  MoveL 10629 to (234.05, 162.02, 144.49) mm, rotated rx 180 ry 0 rz 180 deg; joints [-145.976, -74.933, -32.212, 66.411, 37.63, -61.13]
  Call Extruder(657.74297)
  MoveL 10630 to (233.75, 162.2, 144.49) mm, rotated rx -180 ry 0 rz 180 deg; joints [-145.947, -74.903, -32.271, 66.399, 37.667, -61.104]
  MoveL 10631 to (233.75, 162.2, 144.49) mm, rotated rx -180 ry 0 rz 180 deg; joints [-145.947, -74.903, -32.271, 66.399, 37.667, -61.104]
  Call Extruder(657.94993)
  MoveL 10632 to (233.45, 162.37, 144.49) mm, rotated rx 180 ry 0 rz 180 deg; joints [-145.919, -74.874, -32.33, 66.387, 37.703, -61.078]
  MoveL 10633 to (233.45, 162.37, 144.49) mm, rotated rx 180 ry 0 rz 180 deg; joints [-145.919, -74.874, -32.33, 66.387, 37.703, -61.078]
  Call Extruder(658.15610)
  MoveL 10634 to (233.14, 162.55, 144.49) mm, rotated rx 180 ry 0 rz 180 deg; joints [-145.89, -74.844, -32.388, 66.376, 37.74, -61.053]
  MoveL 10635 to (233.14, 162.55, 144.49) mm, rotated rx 180 ry 0 rz 180 deg; joints [-145.89, -74.844, -32.388, 66.376, 37.74, -61.053]
  Call Extruder(658.33777)
  MoveL 10636 to (232.87, 162.69, 144.49) mm, rotated rx 180 ry 0 rz 180 deg; joints [-145.866, -74.815, -32.446, 66.361, 37.772, -61.026]
  MoveL 10637 to (232.87, 162.69, 144.49) mm, rotated rx 180 ry 0 rz 180 deg; joints [-145.866, -74.815, -32.446, 66.361, 37.772, -61.026]
  Call Extruder(658.49574)
  MoveL 10638 to (232.62, 162.8, 144.49) mm, rotated rx -180 ry 0 rz -180 deg; joints [-145.845, -74.787, -32.501, 66.345, 37.801, -60.997]
  MoveL 10639 to (232.62, 162.8, 144.49) mm, rotated rx -180 ry 0 rz -180 deg; joints [-145.845, -74.787, -32.501, 66.345, 37.801, -60.997]
  Call Extruder(658.65309)
  MoveL 10640 to (232.37, 162.91, 144.49) mm, rotated rx -180 ry 0 rz 180 deg; joints [-145.825, -74.759, -32.557, 66.329, 37.83, -60.969]
  MoveL 10641 to (232.37, 162.91, 144.49) mm, rotated rx -180 ry 0 rz 180 deg; joints [-145.825, -74.759, -32.557, 66.329, 37.83, -60.969]
  Call Extruder(658.83583)
  MoveL 10642 to (232.07, 163.02, 144.49) mm, rotated rx 180 ry 0 rz 180 deg; joints [-145.801, -74.725, -32.623, 66.309, 37.864, -60.935]
  MoveL 10643 to (232.07, 163.02, 144.49) mm, rotated rx 180 ry 0 rz 180 deg; joints [-145.801, -74.725, -32.623, 66.309, 37.864, -60.935]
  Call Extruder(659.01781)
  MoveL 10644 to (231.78, 163.15, 144.49) mm, rotated rx -180 ry 0 rz 180 deg; joints [-145.777, -74.692, -32.689, 66.29, 37.898, -60.901]
  MoveL 10645 to (231.78, 163.15, 144.49) mm, rotated rx -180 ry 0 rz 180 deg; joints [-145.777, -74.692, -32.689, 66.29, 37.898, -60.901]
  Call Extruder(659.16515)
  MoveL 10646 to (231.54, 163.24, 144.49) mm, rotated rx -180 ry 0 rz -180 deg; joints [-145.759, -74.664, -32.745, 66.272, 37.926, -60.872]
  MoveL 10647 to (231.54, 163.24, 144.49) mm, rotated rx -180 ry 0 rz -180 deg; joints [-145.759, -74.664, -32.745, 66.272, 37.926, -60.872]
  Call Extruder(659.27837)
  MoveL 10648 to (231.35, 163.3, 144.49) mm, rotated rx -180 ry 0 rz 180 deg; joints [-145.744, -74.641, -32.791, 66.257, 37.947, -60.847]
  MoveL 10649 to (231.35, 163.3, 144.49) mm, rotated rx -180 ry 0 rz 180 deg; joints [-145.744, -74.641, -32.791, 66.257, 37.947, -60.847]
  Call Extruder(659.39115)
  MoveL 10650 to (231.17, 163.36, 144.49) mm, rotated rx 180 ry 0 rz 180 deg; joints [-145.73, -74.618, -32.836, 66.241, 37.969, -60.822]
  MoveL 10651 to (231.17, 163.36, 144.49) mm, rotated rx 180 ry 0 rz 180 deg; joints [-145.73, -74.618, -32.836, 66.241, 37.969, -60.822]
  Call Extruder(659.50349)
  MoveL 10652 to (230.98, 163.42, 144.49) mm, rotated rx 180 ry 0 rz 180 deg; joints [-145.716, -74.594, -32.882, 66.226, 37.99, -60.797]
  MoveL 10653 to (230.98, 163.42, 144.49) mm, rotated rx 180 ry 0 rz 180 deg; joints [-145.716, -74.594, -32.882, 66.226, 37.99, -60.797]
  Call Extruder(659.61538)
  MoveL 10654 to (230.79, 163.48, 144.49) mm, rotated rx 180 ry 0 rz 180 deg; joints [-145.702, -74.571, -32.928, 66.21, 38.012, -60.772]
  MoveL 10655 to (230.79, 163.48, 144.49) mm, rotated rx 180 ry 0 rz 180 deg; joints [-145.702, -74.571, -32.928, 66.21, 38.012, -60.772]
  Call Extruder(659.73678)
  MoveL 10656 to (230.58, 163.55, 144.49) mm, rotated rx 180 ry 0 rz 180 deg; joints [-145.687, -74.546, -32.978, 66.193, 38.035, -60.745]
  MoveL 10657 to (230.58, 163.55, 144.49) mm, rotated rx 180 ry 0 rz 180 deg; joints [-145.687, -74.546, -32.978, 66.193, 38.035, -60.745]
  Call Extruder(659.86760)
  MoveL 10658 to (230.36, 163.61, 144.49) mm, rotated rx 180 ry 0 rz 180 deg; joints [-145.67, -74.518, -33.034, 66.174, 38.06, -60.714]
  MoveL 10659 to (230.36, 163.61, 144.49) mm, rotated rx 180 ry 0 rz 180 deg; joints [-145.67, -74.518, -33.034, 66.174, 38.06, -60.714]
  Call Extruder(659.99784)
  MoveL 10660 to (230.14, 163.68, 144.49) mm, rotated rx 180 ry 0 rz 180 deg; joints [-145.654, -74.49, -33.089, 66.155, 38.086, -60.684]
  MoveL 10661 to (230.14, 163.68, 144.49) mm, rotated rx 180 ry 0 rz 180 deg; joints [-145.654, -74.49, -33.089, 66.155, 38.086, -60.684]
  Call Extruder(660.12753)
  MoveL 10662 to (229.91, 163.75, 144.49) mm, rotated rx 180 ry 0 rz 180 deg; joints [-145.638, -74.462, -33.144, 66.137, 38.111, -60.654]
  MoveL 10663 to (229.91, 163.75, 144.49) mm, rotated rx 180 ry 0 rz 180 deg; joints [-145.638, -74.462, -33.144, 66.137, 38.111, -60.654]
  Call Extruder(660.25665)
  MoveL 10664 to (229.69, 163.82, 144.49) mm, rotated rx -180 ry 0 rz 180 deg; joints [-145.621, -74.434, -33.199, 66.118, 38.136, -60.624]
  MoveL 10665 to (229.69, 163.82, 144.49) mm, rotated rx -180 ry 0 rz 180 deg; joints [-145.621, -74.434, -33.199, 66.118, 38.136, -60.624]
  Call Extruder(660.37172)
  MoveL 10666 to (229.48, 163.86, 144.49) mm, rotated rx 180 ry 0 rz -180 deg; joints [-145.607, -74.407, -33.253, 66.098, 38.159, -60.593]
  MoveL 10667 to (229.48, 163.86, 144.49) mm, rotated rx 180 ry 0 rz -180 deg; joints [-145.607, -74.407, -33.253, 66.098, 38.159, -60.593]
  Call Extruder(660.48634)
  MoveL 10668 to (229.28, 163.91, 144.49) mm, rotated rx 180 ry 0 rz -180 deg; joints [-145.594, -74.38, -33.306, 66.078, 38.182, -60.562]
  MoveL 10669 to (229.28, 163.91, 144.49) mm, rotated rx 180 ry 0 rz -180 deg; joints [-145.594, -74.38, -33.306, 66.078, 38.182, -60.562]
  Call Extruder(660.60051)
  MoveL 10670 to (229.08, 163.95, 144.49) mm, rotated rx 180 ry 0 rz 180 deg; joints [-145.58, -74.353, -33.36, 66.058, 38.204, -60.532]
  MoveL 10671 to (229.08, 163.95, 144.49) mm, rotated rx 180 ry 0 rz 180 deg; joints [-145.58, -74.353, -33.36, 66.058, 38.204, -60.532]
  Call Extruder(660.71423)
  MoveL 10672 to (228.87, 164, 144.49) mm, rotated rx -180 ry 0 rz -180 deg; joints [-145.566, -74.326, -33.414, 66.038, 38.227, -60.501]
  MoveL 10673 to (228.87, 164, 144.49) mm, rotated rx -180 ry 0 rz -180 deg; joints [-145.566, -74.326, -33.414, 66.038, 38.227, -60.501]
  Call Extruder(660.83965)
  MoveL 10674 to (228.65, 164.04, 144.49) mm, rotated rx 180 ry 0 rz -180 deg; joints [-145.551, -74.296, -33.473, 66.016, 38.252, -60.467]
  MoveL 10675 to (228.65, 164.04, 144.49) mm, rotated rx 180 ry 0 rz -180 deg; joints [-145.551, -74.296, -33.473, 66.016, 38.252, -60.467]
  Call Extruder(660.97663)
  MoveL 10676 to (228.4, 164.09, 144.49) mm, rotated rx 180 ry 0 rz 180 deg; joints [-145.535, -74.263, -33.539, 65.991, 38.28, -60.429]
  MoveL 10677 to (228.4, 164.09, 144.49) mm, rotated rx 180 ry 0 rz 180 deg; joints [-145.535, -74.263, -33.539, 65.991, 38.28, -60.429]
  Call Extruder(661.11299)
  MoveL 10678 to (228.15, 164.14, 144.49) mm, rotated rx 180 ry 0 rz 180 deg; joints [-145.518, -74.229, -33.606, 65.966, 38.308, -60.391]
  MoveL 10679 to (228.15, 164.14, 144.49) mm, rotated rx 180 ry 0 rz 180 deg; joints [-145.518, -74.229, -33.606, 65.966, 38.308, -60.391]
  Call Extruder(661.24875)
  MoveL 10680 to (227.9, 164.19, 144.49) mm, rotated rx 180 ry 0 rz 180 deg; joints [-145.502, -74.196, -33.672, 65.942, 38.335, -60.353]
  MoveL 10681 to (227.9, 164.19, 144.49) mm, rotated rx 180 ry 0 rz 180 deg; joints [-145.502, -74.196, -33.672, 65.942, 38.335, -60.353]
  Call Extruder(661.38390)
  MoveL 10682 to (227.65, 164.24, 144.49) mm, rotated rx 180 ry 0 rz -180 deg; joints [-145.485, -74.163, -33.738, 65.917, 38.363, -60.315]
  MoveL 10683 to (227.65, 164.24, 144.49) mm, rotated rx 180 ry 0 rz -180 deg; joints [-145.485, -74.163, -33.738, 65.917, 38.363, -60.315]
  Call Extruder(661.51844)
  MoveL 10684 to (227.4, 164.29, 144.49) mm, rotated rx -180 ry 0 rz 180 deg; joints [-145.469, -74.129, -33.803, 65.893, 38.39, -60.278]
  MoveL 10685 to (227.4, 164.29, 144.49) mm, rotated rx -180 ry 0 rz 180 deg; joints [-145.469, -74.129, -33.803, 65.893, 38.39, -60.278]
  Call Extruder(661.65236)
  MoveL 10686 to (227.15, 164.34, 144.49) mm, rotated rx -180 ry 0 rz -180 deg; joints [-145.453, -74.096, -33.869, 65.868, 38.418, -60.24]
  MoveL 10687 to (227.15, 164.34, 144.49) mm, rotated rx -180 ry 0 rz -180 deg; joints [-145.453, -74.096, -33.869, 65.868, 38.418, -60.24]
  Call Extruder(661.80023)
  MoveL 10688 to (226.87, 164.39, 144.49) mm, rotated rx 180 ry 0 rz -180 deg; joints [-145.435, -74.059, -33.943, 65.84, 38.448, -60.197]
  MoveL 10689 to (226.87, 164.39, 144.49) mm, rotated rx 180 ry 0 rz -180 deg; joints [-145.435, -74.059, -33.943, 65.84, 38.448, -60.197]
  Call Extruder(661.96197)
  MoveL 10690 to (226.57, 164.44, 144.49) mm, rotated rx 180 ry 0 rz 180 deg; joints [-145.415, -74.017, -34.026, 65.809, 38.482, -60.149]
  MoveL 10691 to (226.57, 164.44, 144.49) mm, rotated rx 180 ry 0 rz 180 deg; joints [-145.415, -74.017, -34.026, 65.809, 38.482, -60.149]
  Call Extruder(662.12298)
  MoveL 10692 to (226.26, 164.49, 144.49) mm, rotated rx -180 ry 0 rz 180 deg; joints [-145.396, -73.975, -34.109, 65.777, 38.516, -60.101]
  MoveL 10693 to (226.26, 164.49, 144.49) mm, rotated rx -180 ry 0 rz 180 deg; joints [-145.396, -73.975, -34.109, 65.777, 38.516, -60.101]
  Call Extruder(662.28327)
  MoveL 10694 to (225.95, 164.53, 144.49) mm, rotated rx -180 ry 0 rz 180 deg; joints [-145.377, -73.934, -34.191, 65.746, 38.549, -60.054]
  MoveL 10695 to (225.95, 164.53, 144.49) mm, rotated rx -180 ry 0 rz 180 deg; joints [-145.377, -73.934, -34.191, 65.746, 38.549, -60.054]
  Call Extruder(662.44282)
  MoveL 10696 to (225.65, 164.58, 144.49) mm, rotated rx -180 ry 0 rz 180 deg; joints [-145.357, -73.892, -34.273, 65.715, 38.583, -60.006]
  MoveL 10697 to (225.65, 164.58, 144.49) mm, rotated rx -180 ry 0 rz 180 deg; joints [-145.357, -73.892, -34.273, 65.715, 38.583, -60.006]
  Call Extruder(662.60165)
  MoveL 10698 to (225.34, 164.63, 144.49) mm, rotated rx -180 ry 0 rz 180 deg; joints [-145.338, -73.851, -34.355, 65.684, 38.616, -59.959]
  MoveL 10699 to (225.34, 164.63, 144.49) mm, rotated rx -180 ry 0 rz 180 deg; joints [-145.338, -73.851, -34.355, 65.684, 38.616, -59.959]
  Call Extruder(662.78032)
  MoveL 10700 to (225, 164.68, 144.49) mm, rotated rx 180 ry 0 rz 180 deg; joints [-145.317, -73.803, -34.45, 65.647, 38.654, -59.904]
  MoveL 10701 to (225, 164.68, 144.49) mm, rotated rx 180 ry 0 rz 180 deg; joints [-145.317, -73.803, -34.45, 65.647, 38.654, -59.904]
  Call Extruder(662.97876)
  MoveL 10702 to (224.61, 164.72, 144.49) mm, rotated rx -180 ry 0 rz 180 deg; joints [-145.293, -73.749, -34.557, 65.606, 38.696, -59.841]
  MoveL 10703 to (224.61, 164.72, 144.49) mm, rotated rx -180 ry 0 rz 180 deg; joints [-145.293, -73.749, -34.557, 65.606, 38.696, -59.841]
  Call Extruder(663.17634)
  MoveL 10704 to (224.22, 164.77, 144.49) mm, rotated rx 180 ry 0 rz 180 deg; joints [-145.27, -73.696, -34.664, 65.565, 38.738, -59.779]
  MoveL 10705 to (224.22, 164.77, 144.49) mm, rotated rx 180 ry 0 rz 180 deg; joints [-145.27, -73.696, -34.664, 65.565, 38.738, -59.779]
  Call Extruder(663.37305)
  MoveL 10706 to (223.83, 164.82, 144.49) mm, rotated rx 180 ry 0 rz 180 deg; joints [-145.246, -73.642, -34.77, 65.524, 38.78, -59.717]
  MoveL 10707 to (223.83, 164.82, 144.49) mm, rotated rx 180 ry 0 rz 180 deg; joints [-145.246, -73.642, -34.77, 65.524, 38.78, -59.717]
  Call Extruder(663.56888)
  MoveL 10708 to (223.45, 164.86, 144.49) mm, rotated rx 180 ry 0 rz 180 deg; joints [-145.223, -73.588, -34.876, 65.483, 38.823, -59.655]
  MoveL 10709 to (223.45, 164.86, 144.49) mm, rotated rx 180 ry 0 rz 180 deg; joints [-145.223, -73.588, -34.876, 65.483, 38.823, -59.655]
  Call Extruder(663.86424)
  MoveL 10710 to (222.86, 164.91, 144.49) mm, rotated rx 180 ry 0 rz -180 deg; joints [-145.189, -73.505, -35.042, 65.418, 38.886, -59.557]
  MoveL 10711 to (222.86, 164.91, 144.49) mm, rotated rx 180 ry 0 rz -180 deg; joints [-145.189, -73.505, -35.042, 65.418, 38.886, -59.557]
  Call Extruder(664.15827)
  MoveL 10712 to (222.27, 164.95, 144.49) mm, rotated rx 180 ry 0 rz 180 deg; joints [-145.155, -73.422, -35.207, 65.353, 38.949, -59.46]
  MoveL 10713 to (222.27, 164.95, 144.49) mm, rotated rx 180 ry 0 rz 180 deg; joints [-145.155, -73.422, -35.207, 65.353, 38.949, -59.46]
  Call Extruder(664.45096)
  MoveL 10714 to (221.68, 165, 144.49) mm, rotated rx 180 ry 0 rz 180 deg; joints [-145.121, -73.339, -35.371, 65.289, 39.013, -59.364]
  MoveL 10715 to (221.68, 165, 144.49) mm, rotated rx 180 ry 0 rz 180 deg; joints [-145.121, -73.339, -35.371, 65.289, 39.013, -59.364]
  Call Extruder(665.02441)
  MoveL 10716 to (220.52, 165.05, 144.49) mm, rotated rx 180 ry 0 rz 180 deg; joints [-145.056, -73.172, -35.703, 65.157, 39.137, -59.167]
  MoveL 10717 to (220.52, 165.05, 144.49) mm, rotated rx 180 ry 0 rz 180 deg; joints [-145.056, -73.172, -35.703, 65.157, 39.137, -59.167]
  Call Extruder(665.73842)
  MoveL 10718 to (219.06, 165.09, 144.49) mm, rotated rx 180 ry 0 rz 180 deg; joints [-144.977, -72.963, -36.118, 64.992, 39.292, -58.921]
  Call Extruder(782.58519)
  MoveL 10719 to (-19.06, 165.09, 144.49) mm, rotated rx -180 ry 0 rz 180 deg; joints [-127.435, -51.662, -80.11, 62.98, 63.042, -41.636]
  Call Extruder(783.01380)
  MoveL 10720 to (-19.94, 165.07, 144.49) mm, rotated rx 180 ry 0 rz 180 deg; joints [-127.348, -51.612, -80.219, 63.026, 63.126, -41.61]
  MoveL 10721 to (-19.94, 165.07, 144.49) mm, rotated rx 180 ry 0 rz 180 deg; joints [-127.348, -51.612, -80.219, 63.026, 63.126, -41.61]
  Call Extruder(783.58725)
  MoveL 10722 to (-21.1, 165.02, 144.49) mm, rotated rx -180 ry 0 rz 180 deg; joints [-127.235, -51.545, -80.367, 63.085, 63.238, -41.573]
  MoveL 10723 to (-21.1, 165.02, 144.49) mm, rotated rx -180 ry 0 rz 180 deg; joints [-127.235, -51.545, -80.367, 63.085, 63.238, -41.573]
  Call Extruder(784.02155)
  MoveL 10724 to (-21.97, 164.98, 144.49) mm, rotated rx 180 ry 0 rz 180 deg; joints [-127.15, -51.493, -80.48, 63.129, 63.322, -41.543]
  MoveL 10725 to (-21.97, 164.98, 144.49) mm, rotated rx 180 ry 0 rz 180 deg; joints [-127.15, -51.493, -80.48, 63.129, 63.322, -41.543]
  Call Extruder(784.31557)
  MoveL 10726 to (-22.56, 164.93, 144.49) mm, rotated rx 180 ry 0 rz 180 deg; joints [-127.093, -51.457, -80.558, 63.157, 63.378, -41.522]
  MoveL 10727 to (-22.56, 164.93, 144.49) mm, rotated rx 180 ry 0 rz 180 deg; joints [-127.093, -51.457, -80.558, 63.157, 63.378, -41.522]
  Call Extruder(784.61093)
  MoveL 10728 to (-23.15, 164.89, 144.49) mm, rotated rx 180 ry 0 rz 180 deg; joints [-127.037, -51.421, -80.636, 63.185, 63.435, -41.501]
  MoveL 10729 to (-23.15, 164.89, 144.49) mm, rotated rx 180 ry 0 rz 180 deg; joints [-127.037, -51.421, -80.636, 63.185, 63.435, -41.501]
  Call Extruder(784.85715)
  MoveL 10730 to (-23.64, 164.84, 144.49) mm, rotated rx 180 ry 0 rz 180 deg; joints [-126.991, -51.391, -80.702, 63.207, 63.481, -41.482]
  MoveL 10731 to (-23.64, 164.84, 144.49) mm, rotated rx 180 ry 0 rz 180 deg; joints [-126.991, -51.391, -80.702, 63.207, 63.481, -41.482]
  Call Extruder(785.05385)
  MoveL 10732 to (-24.03, 164.79, 144.49) mm, rotated rx -180 ry 0 rz 180 deg; joints [-126.955, -51.367, -80.756, 63.224, 63.518, -41.467]
  MoveL 10733 to (-24.03, 164.79, 144.49) mm, rotated rx -180 ry 0 rz 180 deg; joints [-126.955, -51.367, -80.756, 63.224, 63.518, -41.467]
  Call Extruder(785.25143)
  MoveL 10734 to (-24.42, 164.75, 144.49) mm, rotated rx -180 ry 0 rz 180 deg; joints [-126.919, -51.342, -80.81, 63.242, 63.555, -41.451]
  MoveL 10735 to (-24.42, 164.75, 144.49) mm, rotated rx -180 ry 0 rz 180 deg; joints [-126.919, -51.342, -80.81, 63.242, 63.555, -41.451]
  Call Extruder(785.44987)
  MoveL 10736 to (-24.8, 164.7, 144.49) mm, rotated rx -180 ry 0 rz 180 deg; joints [-126.883, -51.318, -80.863, 63.259, 63.592, -41.435]
  MoveL 10737 to (-24.8, 164.7, 144.49) mm, rotated rx -180 ry 0 rz 180 deg; joints [-126.883, -51.318, -80.863, 63.259, 63.592, -41.435]
  Call Extruder(785.64918)
  MoveL 10738 to (-25.19, 164.66, 144.49) mm, rotated rx 180 ry 0 rz 180 deg; joints [-126.847, -51.293, -80.917, 63.276, 63.629, -41.42]
  MoveL 10739 to (-25.19, 164.66, 144.49) mm, rotated rx 180 ry 0 rz 180 deg; joints [-126.847, -51.293, -80.917, 63.276, 63.629, -41.42]
  Call Extruder(785.80801)
  MoveL 10740 to (-25.5, 164.61, 144.49) mm, rotated rx -180 ry 0 rz 180 deg; joints [-126.82, -51.273, -80.961, 63.288, 63.658, -41.406]
  MoveL 10741 to (-25.5, 164.61, 144.49) mm, rotated rx -180 ry 0 rz 180 deg; joints [-126.82, -51.273, -80.961, 63.288, 63.658, -41.406]
  Call Extruder(785.96757)
  MoveL 10742 to (-25.8, 164.56, 144.49) mm, rotated rx 180 ry 0 rz 180 deg; joints [-126.792, -51.253, -81.005, 63.301, 63.687, -41.393]
  MoveL 10743 to (-25.8, 164.56, 144.49) mm, rotated rx 180 ry 0 rz 180 deg; joints [-126.792, -51.253, -81.005, 63.301, 63.687, -41.393]
  Call Extruder(786.12786)
  MoveL 10744 to (-26.11, 164.51, 144.49) mm, rotated rx 180 ry 0 rz -180 deg; joints [-126.765, -51.233, -81.049, 63.313, 63.716, -41.379]
  MoveL 10745 to (-26.11, 164.51, 144.49) mm, rotated rx 180 ry 0 rz -180 deg; joints [-126.765, -51.233, -81.049, 63.313, 63.716, -41.379]
  Call Extruder(786.28887)
  MoveL 10746 to (-26.41, 164.46, 144.49) mm, rotated rx -180 ry 0 rz 180 deg; joints [-126.737, -51.213, -81.093, 63.326, 63.745, -41.365]
  MoveL 10747 to (-26.41, 164.46, 144.49) mm, rotated rx -180 ry 0 rz 180 deg; joints [-126.737, -51.213, -81.093, 63.326, 63.745, -41.365]
  Call Extruder(786.45061)
  MoveL 10748 to (-26.72, 164.41, 144.49) mm, rotated rx 180 ry 0 rz 180 deg; joints [-126.71, -51.193, -81.137, 63.338, 63.774, -41.352]
  MoveL 10749 to (-26.72, 164.41, 144.49) mm, rotated rx 180 ry 0 rz 180 deg; joints [-126.71, -51.193, -81.137, 63.338, 63.774, -41.352]
  Call Extruder(786.61308)
  MoveL 10750 to (-27.03, 164.36, 144.49) mm, rotated rx 180 ry 0 rz 180 deg; joints [-126.682, -51.172, -81.181, 63.351, 63.803, -41.338]
  MoveL 10751 to (-27.03, 164.36, 144.49) mm, rotated rx 180 ry 0 rz 180 deg; joints [-126.682, -51.172, -81.181, 63.351, 63.803, -41.338]
  Call Extruder(786.74701)
  MoveL 10752 to (-27.27, 164.32, 144.49) mm, rotated rx -180 ry 0 rz 180 deg; joints [-126.66, -51.155, -81.218, 63.36, 63.826, -41.326]
  MoveL 10753 to (-27.27, 164.32, 144.49) mm, rotated rx -180 ry 0 rz 180 deg; joints [-126.66, -51.155, -81.218, 63.36, 63.826, -41.326]
  Call Extruder(786.88155)
  MoveL 10754 to (-27.52, 164.27, 144.49) mm, rotated rx -180 ry 0 rz -180 deg; joints [-126.638, -51.138, -81.256, 63.37, 63.85, -41.314]
  MoveL 10755 to (-27.52, 164.27, 144.49) mm, rotated rx -180 ry 0 rz -180 deg; joints [-126.638, -51.138, -81.256, 63.37, 63.85, -41.314]
  Call Extruder(787.01669)
  MoveL 10756 to (-27.77, 164.22, 144.49) mm, rotated rx -180 ry 0 rz 180 deg; joints [-126.617, -51.121, -81.293, 63.379, 63.873, -41.301]
  MoveL 10757 to (-27.77, 164.22, 144.49) mm, rotated rx -180 ry 0 rz 180 deg; joints [-126.617, -51.121, -81.293, 63.379, 63.873, -41.301]
  Call Extruder(787.15245)
  MoveL 10758 to (-28.02, 164.17, 144.49) mm, rotated rx 180 ry 0 rz 180 deg; joints [-126.595, -51.104, -81.33, 63.388, 63.897, -41.289]
  MoveL 10759 to (-28.02, 164.17, 144.49) mm, rotated rx 180 ry 0 rz 180 deg; joints [-126.595, -51.104, -81.33, 63.388, 63.897, -41.289]
  Call Extruder(787.28882)
  MoveL 10760 to (-28.27, 164.12, 144.49) mm, rotated rx -180 ry 0 rz -180 deg; joints [-126.573, -51.087, -81.368, 63.398, 63.92, -41.277]
  MoveL 10761 to (-28.27, 164.12, 144.49) mm, rotated rx -180 ry 0 rz -180 deg; joints [-126.573, -51.087, -81.368, 63.398, 63.92, -41.277]
  Call Extruder(787.42580)
  MoveL 10762 to (-28.52, 164.07, 144.49) mm, rotated rx -180 ry 0 rz -180 deg; joints [-126.551, -51.07, -81.405, 63.407, 63.944, -41.265]
  MoveL 10763 to (-28.52, 164.07, 144.49) mm, rotated rx -180 ry 0 rz -180 deg; joints [-126.551, -51.07, -81.405, 63.407, 63.944, -41.265]
  Call Extruder(787.56338)
  MoveL 10764 to (-28.77, 164.02, 144.49) mm, rotated rx 180 ry 0 rz -180 deg; joints [-126.529, -51.053, -81.442, 63.417, 63.967, -41.253]
  MoveL 10765 to (-28.77, 164.02, 144.49) mm, rotated rx 180 ry 0 rz -180 deg; joints [-126.529, -51.053, -81.442, 63.417, 63.967, -41.253]
  Call Extruder(787.67710)
  MoveL 10766 to (-28.97, 163.97, 144.49) mm, rotated rx -180 ry 0 rz 180 deg; joints [-126.511, -51.039, -81.473, 63.424, 63.987, -41.243]
  MoveL 10767 to (-28.97, 163.97, 144.49) mm, rotated rx -180 ry 0 rz 180 deg; joints [-126.511, -51.039, -81.473, 63.424, 63.987, -41.243]
  Call Extruder(787.79127)
  MoveL 10768 to (-29.18, 163.93, 144.49) mm, rotated rx -180 ry 0 rz -180 deg; joints [-126.494, -51.025, -81.504, 63.431, 64.006, -41.232]
  MoveL 10769 to (-29.18, 163.93, 144.49) mm, rotated rx -180 ry 0 rz -180 deg; joints [-126.494, -51.025, -81.504, 63.431, 64.006, -41.232]
  Call Extruder(787.90589)
  MoveL 10770 to (-29.38, 163.88, 144.49) mm, rotated rx 180 ry 0 rz 180 deg; joints [-126.476, -51.011, -81.535, 63.439, 64.025, -41.222]
  MoveL 10771 to (-29.38, 163.88, 144.49) mm, rotated rx 180 ry 0 rz 180 deg; joints [-126.476, -51.011, -81.535, 63.439, 64.025, -41.222]
  Call Extruder(788.02096)
  MoveL 10772 to (-29.59, 163.84, 144.49) mm, rotated rx 180 ry 0 rz 180 deg; joints [-126.459, -50.997, -81.566, 63.446, 64.044, -41.211]
  MoveL 10773 to (-29.59, 163.84, 144.49) mm, rotated rx 180 ry 0 rz 180 deg; joints [-126.459, -50.997, -81.566, 63.446, 64.044, -41.211]
  Call Extruder(788.14320)
  MoveL 10774 to (-29.8, 163.78, 144.49) mm, rotated rx -180 ry 0 rz 180 deg; joints [-126.441, -50.981, -81.6, 63.453, 64.064, -41.2]
  MoveL 10775 to (-29.8, 163.78, 144.49) mm, rotated rx -180 ry 0 rz 180 deg; joints [-126.441, -50.981, -81.6, 63.453, 64.064, -41.2]
  Call Extruder(788.27288)
  MoveL 10776 to (-30.02, 163.72, 144.49) mm, rotated rx 180 ry 0 rz -180 deg; joints [-126.423, -50.964, -81.638, 63.459, 64.085, -41.186]
  MoveL 10777 to (-30.02, 163.72, 144.49) mm, rotated rx 180 ry 0 rz -180 deg; joints [-126.423, -50.964, -81.638, 63.459, 64.085, -41.186]
  Call Extruder(788.40312)
  MoveL 10778 to (-30.25, 163.65, 144.49) mm, rotated rx -180 ry 0 rz 180 deg; joints [-126.405, -50.947, -81.675, 63.466, 64.106, -41.173]
  MoveL 10779 to (-30.25, 163.65, 144.49) mm, rotated rx -180 ry 0 rz 180 deg; joints [-126.405, -50.947, -81.675, 63.466, 64.106, -41.173]
  Call Extruder(788.53393)
  MoveL 10780 to (-30.47, 163.58, 144.49) mm, rotated rx 180 ry 0 rz -180 deg; joints [-126.387, -50.931, -81.711, 63.472, 64.127, -41.159]
  MoveL 10781 to (-30.47, 163.58, 144.49) mm, rotated rx 180 ry 0 rz -180 deg; joints [-126.387, -50.931, -81.711, 63.472, 64.127, -41.159]
  Call Extruder(788.66530)
  MoveL 10782 to (-30.69, 163.51, 144.49) mm, rotated rx -180 ry 0 rz -180 deg; joints [-126.369, -50.914, -81.748, 63.478, 64.148, -41.146]
  MoveL 10783 to (-30.69, 163.51, 144.49) mm, rotated rx -180 ry 0 rz -180 deg; joints [-126.369, -50.914, -81.748, 63.478, 64.148, -41.146]
  Call Extruder(788.77719)
  MoveL 10784 to (-30.88, 163.45, 144.49) mm, rotated rx 180 ry 0 rz -180 deg; joints [-126.354, -50.899, -81.78, 63.483, 64.165, -41.134]
  MoveL 10785 to (-30.88, 163.45, 144.49) mm, rotated rx 180 ry 0 rz -180 deg; joints [-126.354, -50.899, -81.78, 63.483, 64.165, -41.134]
  Call Extruder(788.88953)
  MoveL 10786 to (-31.07, 163.39, 144.49) mm, rotated rx 180 ry 0 rz 180 deg; joints [-126.339, -50.885, -81.812, 63.488, 64.183, -41.122]
  MoveL 10787 to (-31.07, 163.39, 144.49) mm, rotated rx 180 ry 0 rz 180 deg; joints [-126.339, -50.885, -81.812, 63.488, 64.183, -41.122]
  Call Extruder(789.00231)
  MoveL 10788 to (-31.26, 163.33, 144.49) mm, rotated rx 180 ry 0 rz 180 deg; joints [-126.324, -50.87, -81.844, 63.493, 64.2, -41.11]
  MoveL 10789 to (-31.26, 163.33, 144.49) mm, rotated rx 180 ry 0 rz 180 deg; joints [-126.324, -50.87, -81.844, 63.493, 64.2, -41.11]
  Call Extruder(789.11553)
  MoveL 10790 to (-31.45, 163.27, 144.49) mm, rotated rx 180 ry 0 rz 180 deg; joints [-126.309, -50.856, -81.875, 63.498, 64.218, -41.099]
  MoveL 10791 to (-31.45, 163.27, 144.49) mm, rotated rx 180 ry 0 rz 180 deg; joints [-126.309, -50.856, -81.875, 63.498, 64.218, -41.099]
  Call Extruder(789.22920)
  MoveL 10792 to (-31.64, 163.21, 144.49) mm, rotated rx -180 ry 0 rz -180 deg; joints [-126.294, -50.842, -81.907, 63.503, 64.235, -41.087]
  MoveL 10793 to (-31.64, 163.21, 144.49) mm, rotated rx -180 ry 0 rz -180 deg; joints [-126.294, -50.842, -81.907, 63.503, 64.235, -41.087]
  Call Extruder(789.41118)
  MoveL 10794 to (-31.93, 163.09, 144.49) mm, rotated rx -180 ry 0 rz 180 deg; joints [-126.273, -50.817, -81.96, 63.508, 64.262, -41.066]
  MoveL 10795 to (-31.93, 163.09, 144.49) mm, rotated rx -180 ry 0 rz 180 deg; joints [-126.273, -50.817, -81.96, 63.508, 64.262, -41.066]
  Call Extruder(789.59392)
  MoveL 10796 to (-32.22, 162.97, 144.49) mm, rotated rx 180 ry 0 rz 180 deg; joints [-126.252, -50.793, -82.014, 63.514, 64.289, -41.045]
  MoveL 10797 to (-32.22, 162.97, 144.49) mm, rotated rx 180 ry 0 rz 180 deg; joints [-126.252, -50.793, -82.014, 63.514, 64.289, -41.045]
  Call Extruder(789.76433)
  MoveL 10798 to (-32.49, 162.85, 144.49) mm, rotated rx -180 ry 0 rz -180 deg; joints [-126.233, -50.771, -82.063, 63.518, 64.314, -41.025]
  MoveL 10799 to (-32.49, 162.85, 144.49) mm, rotated rx -180 ry 0 rz -180 deg; joints [-126.233, -50.771, -82.063, 63.518, 64.314, -41.025]
  Call Extruder(789.92231)
  MoveL 10800 to (-32.74, 162.74, 144.49) mm, rotated rx 180 ry 0 rz -180 deg; joints [-126.215, -50.75, -82.109, 63.522, 64.336, -41.006]
  MoveL 10801 to (-32.74, 162.74, 144.49) mm, rotated rx 180 ry 0 rz -180 deg; joints [-126.215, -50.75, -82.109, 63.522, 64.336, -41.006]
  Call Extruder(790.08088)
  MoveL 10802 to (-32.99, 162.64, 144.49) mm, rotated rx -180 ry 0 rz 180 deg; joints [-126.197, -50.729, -82.155, 63.526, 64.359, -40.988]
  MoveL 10803 to (-32.99, 162.64, 144.49) mm, rotated rx -180 ry 0 rz 180 deg; joints [-126.197, -50.729, -82.155, 63.526, 64.359, -40.988]
  Call Extruder(790.28705)
  MoveL 10804 to (-33.29, 162.46, 144.49) mm, rotated rx 180 ry 0 rz 180 deg; joints [-126.179, -50.7, -82.218, 63.527, 64.387, -40.96]
  MoveL 10805 to (-33.29, 162.46, 144.49) mm, rotated rx 180 ry 0 rz 180 deg; joints [-126.179, -50.7, -82.218, 63.527, 64.387, -40.96]
  Call Extruder(790.49399)
  MoveL 10806 to (-33.6, 162.29, 144.49) mm, rotated rx -180 ry 0 rz 180 deg; joints [-126.16, -50.671, -82.281, 63.528, 64.414, -40.933]
  MoveL 10807 to (-33.6, 162.29, 144.49) mm, rotated rx -180 ry 0 rz 180 deg; joints [-126.16, -50.671, -82.281, 63.528, 64.414, -40.933]
  Call Extruder(790.70172)
  MoveL 10808 to (-33.9, 162.11, 144.49) mm, rotated rx 180 ry 0 rz 180 deg; joints [-126.142, -50.643, -82.344, 63.528, 64.441, -40.905]
  MoveL 10809 to (-33.9, 162.11, 144.49) mm, rotated rx 180 ry 0 rz 180 deg; joints [-126.142, -50.643, -82.344, 63.528, 64.441, -40.905]
  Call Extruder(790.91022)
  MoveL 10810 to (-34.21, 161.94, 144.49) mm, rotated rx -180 ry 0 rz 180 deg; joints [-126.123, -50.614, -82.407, 63.529, 64.469, -40.878]
  MoveL 10811 to (-34.21, 161.94, 144.49) mm, rotated rx -180 ry 0 rz 180 deg; joints [-126.123, -50.614, -82.407, 63.529, 64.469, -40.878]
  Call Extruder(791.08976)
  MoveL 10812 to (-34.45, 161.76, 144.49) mm, rotated rx 180 ry 0 rz -180 deg; joints [-126.111, -50.589, -82.464, 63.526, 64.491, -40.852]
  MoveL 10813 to (-34.45, 161.76, 144.49) mm, rotated rx 180 ry 0 rz -180 deg; joints [-126.111, -50.589, -82.464, 63.526, 64.491, -40.852]
  Call Extruder(791.42319)
  MoveL 10814 to (-34.9, 161.43, 144.49) mm, rotated rx 180 ry 0 rz 180 deg; joints [-126.089, -50.541, -82.568, 63.52, 64.53, -40.804]
  MoveL 10815 to (-34.9, 161.43, 144.49) mm, rotated rx 180 ry 0 rz 180 deg; joints [-126.089, -50.541, -82.568, 63.52, 64.53, -40.804]
  Call Extruder(791.75781)
  MoveL 10816 to (-35.35, 161.1, 144.49) mm, rotated rx -180 ry 0 rz 180 deg; joints [-126.067, -50.494, -82.672, 63.515, 64.57, -40.755]
  Call Extruder(792.58572)
  MoveL 10817 to (-36.39, 160.19, 144.49) mm, rotated rx 180 ry 0 rz -180 deg; joints [-126.027, -50.375, -82.935, 63.487, 64.66, -40.627]
  Call Extruder(793.10708)
  MoveL 10818 to (-36.97, 159.54, 144.49) mm, rotated rx -180 ry 0 rz 180 deg; joints [-126.016, -50.298, -83.104, 63.457, 64.709, -40.539]
  Set speed (130.0 mm/s)
  MoveL 10819 to (-38.97, 156.78, 144.49) mm, rotated rx 180 ry 0 rz 180 deg; joints [-126.016, -49.998, -83.768, 63.304, 64.872, -40.18]
  MoveL 10820 to (-38.97, 156.78, 153.89) mm, rotated rx 180 ry 0 rz 180 deg; joints [-126.016, -48.768, -84.147, 63.664, 64.492, -41.023]
  Call Extruder(791.10708)
  Set speed (40.0 mm/s)
  MoveL 10821 to (-38.97, 156.78, 153.89) mm, rotated rx 180 ry 0 rz 180 deg; joints [-126.016, -48.768, -84.147, 63.664, 64.492, -41.023]
  Call Extruder(0.00000)
  Set speed (130.0 mm/s)
  MoveL 10822 to (-31.64, 163.21, 153.89) mm, rotated rx 180 ry 0 rz -180 deg; joints [-126.294, -49.63, -82.285, 63.867, 63.866, -41.918]
  Call Extruder(2.00000)
  Set speed (40.0 mm/s)
  MoveL 10823 to (-31.64, 163.21, 153.89) mm, rotated rx 180 ry 0 rz -180 deg; joints [-126.294, -49.63, -82.285, 63.867, 63.866, -41.918]
  Set speed (30.0 mm/s)
  MoveL 10824 to (-31.64, 163.21, 153.89) mm, rotated rx 180 ry 0 rz -180 deg; joints [-126.294, -49.63, -82.285, 63.867, 63.866, -41.918]
  Call Extruder(2.18198)
  MoveL 10825 to (-31.93, 163.09, 153.89) mm, rotated rx 180 ry 0 rz 180 deg; joints [-126.273, -49.606, -82.338, 63.872, 63.892, -41.897]
  MoveL 10826 to (-31.93, 163.09, 153.89) mm, rotated rx 180 ry 0 rz 180 deg; joints [-126.273, -49.606, -82.338, 63.872, 63.892, -41.897]
  Call Extruder(2.36471)
  MoveL 10827 to (-32.22, 162.97, 153.89) mm, rotated rx 180 ry 0 rz 180 deg; joints [-126.252, -49.581, -82.391, 63.877, 63.919, -41.876]
  MoveL 10828 to (-32.22, 162.97, 153.89) mm, rotated rx 180 ry 0 rz 180 deg; joints [-126.252, -49.581, -82.391, 63.877, 63.919, -41.876]
  Call Extruder(2.53265)
  MoveL 10829 to (-32.49, 162.85, 153.89) mm, rotated rx 180 ry 0 rz -180 deg; joints [-126.233, -49.558, -82.44, 63.881, 63.943, -41.857]
  MoveL 10830 to (-32.49, 162.85, 153.89) mm, rotated rx 180 ry 0 rz -180 deg; joints [-126.233, -49.558, -82.44, 63.881, 63.943, -41.857]
  Call Extruder(2.68564)
  MoveL 10831 to (-32.73, 162.75, 153.89) mm, rotated rx 180 ry 0 rz 180 deg; joints [-126.216, -49.537, -82.485, 63.885, 63.965, -41.839]
  MoveL 10832 to (-32.73, 162.75, 153.89) mm, rotated rx 180 ry 0 rz 180 deg; joints [-126.216, -49.537, -82.485, 63.885, 63.965, -41.839]
  Call Extruder(2.83919)
  MoveL 10833 to (-32.97, 162.65, 153.89) mm, rotated rx 180 ry 0 rz 180 deg; joints [-126.198, -49.517, -82.529, 63.889, 63.987, -41.822]
  MoveL 10834 to (-32.97, 162.65, 153.89) mm, rotated rx 180 ry 0 rz 180 deg; joints [-126.198, -49.517, -82.529, 63.889, 63.987, -41.822]
  Call Extruder(3.04828)
  MoveL 10835 to (-33.28, 162.47, 153.89) mm, rotated rx -180 ry 0 rz -180 deg; joints [-126.18, -49.487, -82.593, 63.889, 64.015, -41.794]
  MoveL 10836 to (-33.28, 162.47, 153.89) mm, rotated rx -180 ry 0 rz -180 deg; joints [-126.18, -49.487, -82.593, 63.889, 64.015, -41.794]
  Call Extruder(3.25817)
  MoveL 10837 to (-33.59, 162.29, 153.89) mm, rotated rx -180 ry 0 rz -180 deg; joints [-126.161, -49.457, -82.658, 63.89, 64.042, -41.767]
  MoveL 10838 to (-33.59, 162.29, 153.89) mm, rotated rx -180 ry 0 rz -180 deg; joints [-126.161, -49.457, -82.658, 63.89, 64.042, -41.767]
  Call Extruder(3.46884)
  MoveL 10839 to (-33.89, 162.11, 153.89) mm, rotated rx -180 ry 0 rz 180 deg; joints [-126.143, -49.428, -82.722, 63.89, 64.07, -41.739]
  MoveL 10840 to (-33.89, 162.11, 153.89) mm, rotated rx -180 ry 0 rz 180 deg; joints [-126.143, -49.428, -82.722, 63.89, 64.07, -41.739]
  Call Extruder(3.68030)
  MoveL 10841 to (-34.2, 161.93, 153.89) mm, rotated rx -180 ry 0 rz 180 deg; joints [-126.124, -49.398, -82.786, 63.89, 64.097, -41.712]
  MoveL 10842 to (-34.2, 161.93, 153.89) mm, rotated rx -180 ry 0 rz 180 deg; joints [-126.124, -49.398, -82.786, 63.89, 64.097, -41.712]
  Call Extruder(3.88506)
  MoveL 10843 to (-34.48, 161.73, 153.89) mm, rotated rx 180 ry 0 rz -180 deg; joints [-126.11, -49.368, -82.849, 63.888, 64.122, -41.683]
  MoveL 10844 to (-34.48, 161.73, 153.89) mm, rotated rx 180 ry 0 rz -180 deg; joints [-126.11, -49.368, -82.849, 63.888, 64.122, -41.683]
  Call Extruder(4.20602)
  MoveL 10845 to (-34.92, 161.42, 153.89) mm, rotated rx -180 ry 0 rz -180 deg; joints [-126.088, -49.322, -82.95, 63.882, 64.16, -41.637]
  MoveL 10846 to (-34.92, 161.42, 153.89) mm, rotated rx -180 ry 0 rz -180 deg; joints [-126.088, -49.322, -82.95, 63.882, 64.16, -41.637]
  Call Extruder(4.52807)
  MoveL 10847 to (-35.35, 161.1, 153.89) mm, rotated rx 180 ry 0 rz 180 deg; joints [-126.067, -49.275, -83.05, 63.876, 64.198, -41.591]
  Call Extruder(5.35599)
  MoveL 10848 to (-36.39, 160.19, 153.89) mm, rotated rx 180 ry 0 rz -180 deg; joints [-126.027, -49.153, -83.314, 63.848, 64.286, -41.464]
  Call Extruder(6.18392)
  MoveL 10849 to (-37.3, 159.15, 153.89) mm, rotated rx -180 ry 0 rz -180 deg; joints [-126.011, -49.029, -83.582, 63.799, 64.361, -41.326]
  Call Extruder(6.34862)
  MoveL 10850 to (-37.46, 158.93, 153.89) mm, rotated rx 180 ry 0 rz 180 deg; joints [-126.011, -49.004, -83.636, 63.787, 64.374, -41.298]
  MoveL 10851 to (-37.46, 158.93, 153.89) mm, rotated rx 180 ry 0 rz 180 deg; joints [-126.011, -49.004, -83.636, 63.787, 64.374, -41.298]
  Call Extruder(6.67688)
  MoveL 10852 to (-37.79, 158.49, 153.89) mm, rotated rx 180 ry 0 rz 180 deg; joints [-126.011, -48.954, -83.743, 63.762, 64.399, -41.24]
  MoveL 10853 to (-37.79, 158.49, 153.89) mm, rotated rx 180 ry 0 rz 180 deg; joints [-126.011, -48.954, -83.743, 63.762, 64.399, -41.24]
  Call Extruder(7.00398)
  MoveL 10854 to (-38.11, 158.04, 153.89) mm, rotated rx 180 ry 0 rz 180 deg; joints [-126.011, -48.905, -83.85, 63.737, 64.425, -41.183]
  MoveL 10855 to (-38.11, 158.04, 153.89) mm, rotated rx 180 ry 0 rz 180 deg; joints [-126.011, -48.905, -83.85, 63.737, 64.425, -41.183]
  Call Extruder(7.13851)
  MoveL 10856 to (-38.22, 157.85, 153.89) mm, rotated rx 180 ry 0 rz 180 deg; joints [-126.014, -48.885, -83.894, 63.725, 64.433, -41.159]
  MoveL 10857 to (-38.22, 157.85, 153.89) mm, rotated rx 180 ry 0 rz 180 deg; joints [-126.014, -48.885, -83.894, 63.725, 64.433, -41.159]
  Call Extruder(7.35382)
  MoveL 10858 to (-38.41, 157.53, 153.89) mm, rotated rx 180 ry 0 rz -180 deg; joints [-126.019, -48.852, -83.964, 63.704, 64.447, -41.119]
  MoveL 10859 to (-38.41, 157.53, 153.89) mm, rotated rx 180 ry 0 rz -180 deg; joints [-126.019, -48.852, -83.964, 63.704, 64.447, -41.119]
  Call Extruder(7.56829)
  MoveL 10860 to (-38.59, 157.21, 153.89) mm, rotated rx -180 ry 0 rz 180 deg; joints [-126.024, -48.82, -84.035, 63.684, 64.46, -41.08]
  MoveL 10861 to (-38.59, 157.21, 153.89) mm, rotated rx -180 ry 0 rz 180 deg; joints [-126.024, -48.82, -84.035, 63.684, 64.46, -41.08]
  Call Extruder(7.78192)
  MoveL 10862 to (-38.77, 156.9, 153.89) mm, rotated rx 180 ry 0 rz 180 deg; joints [-126.029, -48.787, -84.105, 63.663, 64.473, -41.04]
  MoveL 10863 to (-38.77, 156.9, 153.89) mm, rotated rx 180 ry 0 rz 180 deg; joints [-126.029, -48.787, -84.105, 63.663, 64.473, -41.04]
  Call Extruder(7.96114)
  MoveL 10864 to (-38.91, 156.63, 153.89) mm, rotated rx 180 ry 0 rz 180 deg; joints [-126.035, -48.76, -84.164, 63.644, 64.483, -41.006]
  MoveL 10865 to (-38.91, 156.63, 153.89) mm, rotated rx 180 ry 0 rz 180 deg; joints [-126.035, -48.76, -84.164, 63.644, 64.483, -41.006]
  Call Extruder(8.10685)
  MoveL 10866 to (-39.01, 156.4, 153.89) mm, rotated rx 180 ry 0 rz 180 deg; joints [-126.043, -48.738, -84.211, 63.627, 64.49, -40.978]
  MoveL 10867 to (-39.01, 156.4, 153.89) mm, rotated rx 180 ry 0 rz 180 deg; joints [-126.043, -48.738, -84.211, 63.627, 64.49, -40.978]
  Call Extruder(8.25205)
  MoveL 10868 to (-39.1, 156.17, 153.89) mm, rotated rx 180 ry 0 rz 180 deg; joints [-126.05, -48.716, -84.259, 63.61, 64.496, -40.951]
  MoveL 10869 to (-39.1, 156.17, 153.89) mm, rotated rx 180 ry 0 rz 180 deg; joints [-126.05, -48.716, -84.259, 63.61, 64.496, -40.951]
  Call Extruder(8.43477)
  MoveL 10870 to (-39.23, 155.87, 153.89) mm, rotated rx -180 ry 0 rz -180 deg; joints [-126.06, -48.689, -84.318, 63.588, 64.504, -40.915]
  MoveL 10871 to (-39.23, 155.87, 153.89) mm, rotated rx -180 ry 0 rz -180 deg; joints [-126.06, -48.689, -84.318, 63.588, 64.504, -40.915]
  Call Extruder(8.61673)
  MoveL 10872 to (-39.35, 155.58, 153.89) mm, rotated rx 180 ry 0 rz 180 deg; joints [-126.07, -48.662, -84.378, 63.566, 64.512, -40.88]
  MoveL 10873 to (-39.35, 155.58, 153.89) mm, rotated rx 180 ry 0 rz 180 deg; joints [-126.07, -48.662, -84.378, 63.566, 64.512, -40.88]
  Call Extruder(8.76407)
  MoveL 10874 to (-39.44, 155.34, 153.89) mm, rotated rx 180 ry 0 rz 180 deg; joints [-126.079, -48.639, -84.426, 63.548, 64.518, -40.851]
  MoveL 10875 to (-39.44, 155.34, 153.89) mm, rotated rx 180 ry 0 rz 180 deg; joints [-126.079, -48.639, -84.426, 63.548, 64.518, -40.851]
  Call Extruder(8.87730)
  MoveL 10876 to (-39.5, 155.15, 153.89) mm, rotated rx 180 ry 0 rz 180 deg; joints [-126.087, -48.622, -84.462, 63.533, 64.521, -40.828]
  MoveL 10877 to (-39.5, 155.15, 153.89) mm, rotated rx 180 ry 0 rz 180 deg; joints [-126.087, -48.622, -84.462, 63.533, 64.521, -40.828]
  Call Extruder(8.99009)
  MoveL 10878 to (-39.56, 154.97, 153.89) mm, rotated rx -180 ry 0 rz 180 deg; joints [-126.095, -48.606, -84.499, 63.518, 64.525, -40.806]
  MoveL 10879 to (-39.56, 154.97, 153.89) mm, rotated rx -180 ry 0 rz 180 deg; joints [-126.095, -48.606, -84.499, 63.518, 64.525, -40.806]
  Call Extruder(9.10244)
  MoveL 10880 to (-39.62, 154.78, 153.89) mm, rotated rx -180 ry 0 rz 180 deg; joints [-126.103, -48.589, -84.535, 63.502, 64.528, -40.784]
  MoveL 10881 to (-39.62, 154.78, 153.89) mm, rotated rx -180 ry 0 rz 180 deg; joints [-126.103, -48.589, -84.535, 63.502, 64.528, -40.784]
  Call Extruder(9.21434)
  MoveL 10882 to (-39.68, 154.59, 153.89) mm, rotated rx 180 ry 0 rz 180 deg; joints [-126.111, -48.572, -84.572, 63.487, 64.531, -40.761]
  MoveL 10883 to (-39.68, 154.59, 153.89) mm, rotated rx 180 ry 0 rz 180 deg; joints [-126.111, -48.572, -84.572, 63.487, 64.531, -40.761]
  Call Extruder(9.33574)
  MoveL 10884 to (-39.75, 154.38, 153.89) mm, rotated rx 180 ry 0 rz -180 deg; joints [-126.12, -48.554, -84.611, 63.47, 64.535, -40.737]
  MoveL 10885 to (-39.75, 154.38, 153.89) mm, rotated rx 180 ry 0 rz -180 deg; joints [-126.12, -48.554, -84.611, 63.47, 64.535, -40.737]
  Call Extruder(9.46653)
  MoveL 10886 to (-39.82, 154.16, 153.89) mm, rotated rx -180 ry 0 rz 180 deg; joints [-126.131, -48.534, -84.654, 63.452, 64.539, -40.71]
  MoveL 10887 to (-39.82, 154.16, 153.89) mm, rotated rx -180 ry 0 rz 180 deg; joints [-126.131, -48.534, -84.654, 63.452, 64.539, -40.71]
  Call Extruder(9.59676)
  MoveL 10888 to (-39.88, 153.94, 153.89) mm, rotated rx 180 ry 0 rz 180 deg; joints [-126.141, -48.515, -84.696, 63.434, 64.542, -40.684]
  MoveL 10889 to (-39.88, 153.94, 153.89) mm, rotated rx 180 ry 0 rz 180 deg; joints [-126.141, -48.515, -84.696, 63.434, 64.542, -40.684]
  Call Extruder(9.72643)
  MoveL 10890 to (-39.95, 153.71, 153.89) mm, rotated rx -180 ry 0 rz -180 deg; joints [-126.151, -48.495, -84.739, 63.415, 64.546, -40.657]
  MoveL 10891 to (-39.95, 153.71, 153.89) mm, rotated rx -180 ry 0 rz -180 deg; joints [-126.151, -48.495, -84.739, 63.415, 64.546, -40.657]
  Call Extruder(9.85553)
  MoveL 10892 to (-40.02, 153.49, 153.89) mm, rotated rx 180 ry 0 rz -180 deg; joints [-126.161, -48.475, -84.782, 63.397, 64.549, -40.631]
  MoveL 10893 to (-40.02, 153.49, 153.89) mm, rotated rx 180 ry 0 rz -180 deg; joints [-126.161, -48.475, -84.782, 63.397, 64.549, -40.631]
  Call Extruder(9.97061)
  MoveL 10894 to (-40.06, 153.28, 153.89) mm, rotated rx -180 ry 0 rz 180 deg; joints [-126.173, -48.458, -84.819, 63.379, 64.551, -40.607]
  MoveL 10895 to (-40.06, 153.28, 153.89) mm, rotated rx -180 ry 0 rz 180 deg; joints [-126.173, -48.458, -84.819, 63.379, 64.551, -40.607]
  Call Extruder(10.08525)
  MoveL 10896 to (-40.11, 153.08, 153.89) mm, rotated rx -180 ry 0 rz -180 deg; joints [-126.184, -48.441, -84.856, 63.361, 64.553, -40.583]
  MoveL 10897 to (-40.11, 153.08, 153.89) mm, rotated rx -180 ry 0 rz -180 deg; joints [-126.184, -48.441, -84.856, 63.361, 64.553, -40.583]
  Call Extruder(10.19943)
  MoveL 10898 to (-40.15, 152.88, 153.89) mm, rotated rx -180 ry 0 rz -180 deg; joints [-126.195, -48.424, -84.892, 63.343, 64.554, -40.559]
  MoveL 10899 to (-40.15, 152.88, 153.89) mm, rotated rx -180 ry 0 rz -180 deg; joints [-126.195, -48.424, -84.892, 63.343, 64.554, -40.559]
  Call Extruder(10.31316)
  MoveL 10900 to (-40.2, 152.67, 153.89) mm, rotated rx 180 ry 0 rz 180 deg; joints [-126.206, -48.407, -84.93, 63.325, 64.556, -40.536]
  MoveL 10901 to (-40.2, 152.67, 153.89) mm, rotated rx 180 ry 0 rz 180 deg; joints [-126.206, -48.407, -84.93, 63.325, 64.556, -40.536]
  Call Extruder(10.43859)
  MoveL 10902 to (-40.24, 152.45, 153.89) mm, rotated rx 180 ry 0 rz 180 deg; joints [-126.219, -48.389, -84.97, 63.305, 64.557, -40.509]
  MoveL 10903 to (-40.24, 152.45, 153.89) mm, rotated rx 180 ry 0 rz 180 deg; joints [-126.219, -48.389, -84.97, 63.305, 64.557, -40.509]
  Call Extruder(10.57556)
  MoveL 10904 to (-40.29, 152.2, 153.89) mm, rotated rx 180 ry 0 rz 180 deg; joints [-126.233, -48.368, -85.015, 63.283, 64.559, -40.48]
  MoveL 10905 to (-40.29, 152.2, 153.89) mm, rotated rx 180 ry 0 rz 180 deg; joints [-126.233, -48.368, -85.015, 63.283, 64.559, -40.48]
  Call Extruder(10.71193)
  MoveL 10906 to (-40.34, 151.95, 153.89) mm, rotated rx 180 ry 0 rz -180 deg; joints [-126.248, -48.348, -85.059, 63.26, 64.56, -40.451]
  MoveL 10907 to (-40.34, 151.95, 153.89) mm, rotated rx 180 ry 0 rz -180 deg; joints [-126.248, -48.348, -85.059, 63.26, 64.56, -40.451]
  Call Extruder(10.84768)
  MoveL 10908 to (-40.39, 151.7, 153.89) mm, rotated rx -180 ry 0 rz -180 deg; joints [-126.262, -48.327, -85.103, 63.238, 64.562, -40.423]
  MoveL 10909 to (-40.39, 151.7, 153.89) mm, rotated rx -180 ry 0 rz -180 deg; joints [-126.262, -48.327, -85.103, 63.238, 64.562, -40.423]
  Call Extruder(10.98283)
  MoveL 10910 to (-40.44, 151.45, 153.89) mm, rotated rx 180 ry 0 rz 180 deg; joints [-126.276, -48.307, -85.148, 63.216, 64.563, -40.394]
  MoveL 10911 to (-40.44, 151.45, 153.89) mm, rotated rx 180 ry 0 rz 180 deg; joints [-126.276, -48.307, -85.148, 63.216, 64.563, -40.394]
  Call Extruder(11.11736)
  MoveL 10912 to (-40.49, 151.2, 153.89) mm, rotated rx -180 ry 0 rz -180 deg; joints [-126.291, -48.286, -85.192, 63.194, 64.565, -40.365]
  MoveL 10913 to (-40.49, 151.2, 153.89) mm, rotated rx -180 ry 0 rz -180 deg; joints [-126.291, -48.286, -85.192, 63.194, 64.565, -40.365]
  Call Extruder(11.25129)
  MoveL 10914 to (-40.54, 150.95, 153.89) mm, rotated rx 180 ry 0 rz 180 deg; joints [-126.305, -48.266, -85.236, 63.171, 64.566, -40.336]
  MoveL 10915 to (-40.54, 150.95, 153.89) mm, rotated rx 180 ry 0 rz 180 deg; joints [-126.305, -48.266, -85.236, 63.171, 64.566, -40.336]
  Call Extruder(11.39914)
  MoveL 10916 to (-40.59, 150.67, 153.89) mm, rotated rx -180 ry 0 rz 180 deg; joints [-126.322, -48.244, -85.285, 63.146, 64.567, -40.304]
  MoveL 10917 to (-40.59, 150.67, 153.89) mm, rotated rx -180 ry 0 rz 180 deg; joints [-126.322, -48.244, -85.285, 63.146, 64.567, -40.304]
  Call Extruder(11.56087)
  MoveL 10918 to (-40.64, 150.37, 153.89) mm, rotated rx -180 ry 0 rz 180 deg; joints [-126.341, -48.219, -85.338, 63.118, 64.568, -40.269]
  MoveL 10919 to (-40.64, 150.37, 153.89) mm, rotated rx -180 ry 0 rz 180 deg; joints [-126.341, -48.219, -85.338, 63.118, 64.568, -40.269]
  Call Extruder(11.72186)
  MoveL 10920 to (-40.69, 150.06, 153.89) mm, rotated rx 180 ry 0 rz 180 deg; joints [-126.36, -48.195, -85.391, 63.09, 64.569, -40.234]
  MoveL 10921 to (-40.69, 150.06, 153.89) mm, rotated rx 180 ry 0 rz 180 deg; joints [-126.36, -48.195, -85.391, 63.09, 64.569, -40.234]
  Call Extruder(11.88213)
  MoveL 10922 to (-40.73, 149.76, 153.89) mm, rotated rx 180 ry 0 rz 180 deg; joints [-126.379, -48.171, -85.444, 63.062, 64.569, -40.199]
  MoveL 10923 to (-40.73, 149.76, 153.89) mm, rotated rx 180 ry 0 rz 180 deg; joints [-126.379, -48.171, -85.444, 63.062, 64.569, -40.199]
  Call Extruder(12.04168)
  MoveL 10924 to (-40.78, 149.45, 153.89) mm, rotated rx -180 ry 0 rz 180 deg; joints [-126.398, -48.147, -85.496, 63.034, 64.57, -40.164]
  MoveL 10925 to (-40.78, 149.45, 153.89) mm, rotated rx -180 ry 0 rz 180 deg; joints [-126.398, -48.147, -85.496, 63.034, 64.57, -40.164]
  Call Extruder(12.20049)
  MoveL 10926 to (-40.83, 149.14, 153.89) mm, rotated rx -180 ry 0 rz 180 deg; joints [-126.417, -48.122, -85.549, 63.005, 64.571, -40.129]
  MoveL 10927 to (-40.83, 149.14, 153.89) mm, rotated rx -180 ry 0 rz 180 deg; joints [-126.417, -48.122, -85.549, 63.005, 64.571, -40.129]
  Call Extruder(12.37915)
  MoveL 10928 to (-40.88, 148.8, 153.89) mm, rotated rx -180 ry 0 rz 180 deg; joints [-126.439, -48.095, -85.608, 62.973, 64.571, -40.089]
  MoveL 10929 to (-40.88, 148.8, 153.89) mm, rotated rx -180 ry 0 rz 180 deg; joints [-126.439, -48.095, -85.608, 62.973, 64.571, -40.089]
  Call Extruder(12.57759)
  MoveL 10930 to (-40.92, 148.41, 153.89) mm, rotated rx -180 ry 0 rz 180 deg; joints [-126.465, -48.065, -85.673, 62.936, 64.57, -40.045]
  MoveL 10931 to (-40.92, 148.41, 153.89) mm, rotated rx -180 ry 0 rz 180 deg; joints [-126.465, -48.065, -85.673, 62.936, 64.57, -40.045]
  Call Extruder(12.77517)
  MoveL 10932 to (-40.97, 148.02, 153.89) mm, rotated rx -180 ry 0 rz -180 deg; joints [-126.491, -48.036, -85.738, 62.899, 64.569, -40.001]
  MoveL 10933 to (-40.97, 148.02, 153.89) mm, rotated rx -180 ry 0 rz -180 deg; joints [-126.491, -48.036, -85.738, 62.899, 64.569, -40.001]
  Call Extruder(12.97187)
  MoveL 10934 to (-41.02, 147.63, 153.89) mm, rotated rx 180 ry 0 rz 180 deg; joints [-126.517, -48.006, -85.803, 62.862, 64.569, -39.957]
  MoveL 10935 to (-41.02, 147.63, 153.89) mm, rotated rx 180 ry 0 rz 180 deg; joints [-126.517, -48.006, -85.803, 62.862, 64.569, -39.957]
  Call Extruder(13.16771)
  MoveL 10936 to (-41.06, 147.25, 153.89) mm, rotated rx 180 ry 0 rz 180 deg; joints [-126.543, -47.976, -85.868, 62.825, 64.568, -39.912]
  MoveL 10937 to (-41.06, 147.25, 153.89) mm, rotated rx 180 ry 0 rz 180 deg; joints [-126.543, -47.976, -85.868, 62.825, 64.568, -39.912]
  Call Extruder(13.46311)
  MoveL 10938 to (-41.11, 146.66, 153.89) mm, rotated rx -180 ry 0 rz 180 deg; joints [-126.585, -47.932, -85.964, 62.767, 64.565, -39.846]
  MoveL 10939 to (-41.11, 146.66, 153.89) mm, rotated rx -180 ry 0 rz 180 deg; joints [-126.585, -47.932, -85.964, 62.767, 64.565, -39.846]
  Call Extruder(13.75718)
  MoveL 10940 to (-41.15, 146.07, 153.89) mm, rotated rx -180 ry 0 rz 180 deg; joints [-126.628, -47.888, -86.06, 62.709, 64.561, -39.779]
  MoveL 10941 to (-41.15, 146.07, 153.89) mm, rotated rx -180 ry 0 rz 180 deg; joints [-126.628, -47.888, -86.06, 62.709, 64.561, -39.779]
  Call Extruder(14.04991)
  MoveL 10942 to (-41.2, 145.48, 153.89) mm, rotated rx 180 ry 0 rz 180 deg; joints [-126.67, -47.844, -86.156, 62.651, 64.558, -39.713]
  MoveL 10943 to (-41.2, 145.48, 153.89) mm, rotated rx 180 ry 0 rz 180 deg; joints [-126.67, -47.844, -86.156, 62.651, 64.558, -39.713]
  Call Extruder(14.62336)
  MoveL 10944 to (-41.25, 144.32, 153.89) mm, rotated rx -180 ry 0 rz -180 deg; joints [-126.759, -47.76, -86.339, 62.533, 64.547, -39.583]
  MoveL 10945 to (-41.25, 144.32, 153.89) mm, rotated rx -180 ry 0 rz -180 deg; joints [-126.759, -47.76, -86.339, 62.533, 64.547, -39.583]
  Call Extruder(15.33742)
  MoveL 10946 to (-41.29, 142.86, 153.89) mm, rotated rx -180 ry 0 rz 180 deg; joints [-126.873, -47.657, -86.565, 62.384, 64.531, -39.42]
  Call Extruder(57.40821)
  MoveL 10947 to (-41.29, 57.14, 153.89) mm, rotated rx 180 ry 0 rz 180 deg; joints [-135.148, -42.39, -98.396, 52.089, 63.371, -29.921]
  Call Extruder(57.85446)
  MoveL 10948 to (-41.27, 56.23, 153.89) mm, rotated rx 180 ry 0 rz -180 deg; joints [-135.254, -42.342, -98.505, 51.961, 63.357, -29.82]
  MoveL 10949 to (-41.27, 56.23, 153.89) mm, rotated rx 180 ry 0 rz -180 deg; joints [-135.254, -42.342, -98.505, 51.961, 63.357, -29.82]
  Call Extruder(58.44013)
  MoveL 10950 to (-41.22, 55.04, 153.89) mm, rotated rx 180 ry 0 rz -180 deg; joints [-135.395, -42.282, -98.645, 51.793, 63.336, -29.688]
  MoveL 10951 to (-41.22, 55.04, 153.89) mm, rotated rx 180 ry 0 rz -180 deg; joints [-135.395, -42.282, -98.645, 51.793, 63.336, -29.688]
  Call Extruder(58.87777)
  MoveL 10952 to (-41.17, 54.16, 153.89) mm, rotated rx -180 ry 0 rz 180 deg; joints [-135.502, -42.238, -98.748, 51.666, 63.32, -29.59]
  MoveL 10953 to (-41.17, 54.16, 153.89) mm, rotated rx -180 ry 0 rz 180 deg; joints [-135.502, -42.238, -98.748, 51.666, 63.32, -29.59]
  Call Extruder(59.16609)
  MoveL 10954 to (-41.13, 53.58, 153.89) mm, rotated rx 180 ry 0 rz -180 deg; joints [-135.573, -42.21, -98.813, 51.582, 63.307, -29.527]
  MoveL 10955 to (-41.13, 53.58, 153.89) mm, rotated rx 180 ry 0 rz -180 deg; joints [-135.573, -42.21, -98.813, 51.582, 63.307, -29.527]
  Call Extruder(59.45571)
  MoveL 10956 to (-41.08, 53, 153.89) mm, rotated rx 180 ry 0 rz -180 deg; joints [-135.645, -42.182, -98.877, 51.497, 63.295, -29.463]
  MoveL 10957 to (-41.08, 53, 153.89) mm, rotated rx 180 ry 0 rz -180 deg; joints [-135.645, -42.182, -98.877, 51.497, 63.295, -29.463]
  Call Extruder(59.69701)
  MoveL 10958 to (-41.04, 52.53, 153.89) mm, rotated rx 180 ry 0 rz -180 deg; joints [-135.705, -42.16, -98.93, 51.426, 63.284, -29.41]
  MoveL 10959 to (-41.04, 52.53, 153.89) mm, rotated rx 180 ry 0 rz -180 deg; joints [-135.705, -42.16, -98.93, 51.426, 63.284, -29.41]
  Call Extruder(59.88962)
  MoveL 10960 to (-40.99, 52.15, 153.89) mm, rotated rx 180 ry 0 rz 180 deg; joints [-135.754, -42.142, -98.971, 51.37, 63.274, -29.368]
  MoveL 10961 to (-40.99, 52.15, 153.89) mm, rotated rx 180 ry 0 rz 180 deg; joints [-135.754, -42.142, -98.971, 51.37, 63.274, -29.368]
  Call Extruder(60.08307)
  MoveL 10962 to (-40.95, 51.77, 153.89) mm, rotated rx -180 ry 0 rz -180 deg; joints [-135.804, -42.125, -99.011, 51.312, 63.265, -29.326]
  MoveL 10963 to (-40.95, 51.77, 153.89) mm, rotated rx -180 ry 0 rz -180 deg; joints [-135.804, -42.125, -99.011, 51.312, 63.265, -29.326]
  Call Extruder(60.27736)
  MoveL 10964 to (-40.9, 51.39, 153.89) mm, rotated rx 180 ry 0 rz -180 deg; joints [-135.853, -42.108, -99.052, 51.255, 63.255, -29.285]
  MoveL 10965 to (-40.9, 51.39, 153.89) mm, rotated rx 180 ry 0 rz -180 deg; joints [-135.853, -42.108, -99.052, 51.255, 63.255, -29.285]
  Call Extruder(60.47247)
  MoveL 10966 to (-40.86, 51.01, 153.89) mm, rotated rx 180 ry 0 rz 180 deg; joints [-135.902, -42.09, -99.092, 51.198, 63.246, -29.243]
  MoveL 10967 to (-40.86, 51.01, 153.89) mm, rotated rx 180 ry 0 rz 180 deg; joints [-135.902, -42.09, -99.092, 51.198, 63.246, -29.243]
  Call Extruder(60.63128)
  MoveL 10968 to (-40.81, 50.7, 153.89) mm, rotated rx 180 ry 0 rz -180 deg; joints [-135.943, -42.077, -99.123, 51.151, 63.237, -29.209]
  MoveL 10969 to (-40.81, 50.7, 153.89) mm, rotated rx 180 ry 0 rz -180 deg; joints [-135.943, -42.077, -99.123, 51.151, 63.237, -29.209]
  Call Extruder(60.79083)
  MoveL 10970 to (-40.76, 50.4, 153.89) mm, rotated rx 180 ry 0 rz -180 deg; joints [-135.984, -42.064, -99.154, 51.104, 63.228, -29.176]
  MoveL 10971 to (-40.76, 50.4, 153.89) mm, rotated rx 180 ry 0 rz -180 deg; joints [-135.984, -42.064, -99.154, 51.104, 63.228, -29.176]
  Call Extruder(60.95110)
  MoveL 10972 to (-40.71, 50.09, 153.89) mm, rotated rx 180 ry 0 rz 180 deg; joints [-136.025, -42.05, -99.185, 51.057, 63.219, -29.142]
  MoveL 10973 to (-40.71, 50.09, 153.89) mm, rotated rx 180 ry 0 rz 180 deg; joints [-136.025, -42.05, -99.185, 51.057, 63.219, -29.142]
  Call Extruder(61.11209)
  MoveL 10974 to (-40.66, 49.79, 153.89) mm, rotated rx -180 ry 0 rz -180 deg; joints [-136.067, -42.037, -99.216, 51.01, 63.21, -29.109]
  MoveL 10975 to (-40.66, 49.79, 153.89) mm, rotated rx -180 ry 0 rz -180 deg; joints [-136.067, -42.037, -99.216, 51.01, 63.21, -29.109]
  Call Extruder(61.27382)
  MoveL 10976 to (-40.61, 49.48, 153.89) mm, rotated rx 180 ry 0 rz 180 deg; joints [-136.108, -42.024, -99.247, 50.962, 63.201, -29.075]
  MoveL 10977 to (-40.61, 49.48, 153.89) mm, rotated rx 180 ry 0 rz 180 deg; joints [-136.108, -42.024, -99.247, 50.962, 63.201, -29.075]
  Call Extruder(61.43627)
  MoveL 10978 to (-40.56, 49.17, 153.89) mm, rotated rx 180 ry 0 rz -180 deg; joints [-136.149, -42.011, -99.277, 50.915, 63.192, -29.042]
  MoveL 10979 to (-40.56, 49.17, 153.89) mm, rotated rx 180 ry 0 rz -180 deg; joints [-136.149, -42.011, -99.277, 50.915, 63.192, -29.042]
  Call Extruder(61.57020)
  MoveL 10980 to (-40.52, 48.92, 153.89) mm, rotated rx -180 ry 0 rz 180 deg; joints [-136.184, -42.001, -99.301, 50.875, 63.184, -29.014]
  MoveL 10981 to (-40.52, 48.92, 153.89) mm, rotated rx -180 ry 0 rz 180 deg; joints [-136.184, -42.001, -99.301, 50.875, 63.184, -29.014]
  Call Extruder(61.70473)
  MoveL 10982 to (-40.47, 48.68, 153.89) mm, rotated rx 180 ry 0 rz 180 deg; joints [-136.219, -41.99, -99.325, 50.836, 63.175, -28.987]
  MoveL 10983 to (-40.47, 48.68, 153.89) mm, rotated rx 180 ry 0 rz 180 deg; joints [-136.219, -41.99, -99.325, 50.836, 63.175, -28.987]
  Call Extruder(61.83988)
  MoveL 10984 to (-40.42, 48.43, 153.89) mm, rotated rx 180 ry 0 rz 180 deg; joints [-136.254, -41.98, -99.349, 50.796, 63.167, -28.96]
  MoveL 10985 to (-40.42, 48.43, 153.89) mm, rotated rx 180 ry 0 rz 180 deg; joints [-136.254, -41.98, -99.349, 50.796, 63.167, -28.96]
  Call Extruder(61.97563)
  MoveL 10986 to (-40.37, 48.18, 153.89) mm, rotated rx 180 ry 0 rz -180 deg; joints [-136.288, -41.97, -99.373, 50.757, 63.159, -28.933]
  MoveL 10987 to (-40.37, 48.18, 153.89) mm, rotated rx 180 ry 0 rz -180 deg; joints [-136.288, -41.97, -99.373, 50.757, 63.159, -28.933]
  Call Extruder(62.11200)
  MoveL 10988 to (-40.32, 47.93, 153.89) mm, rotated rx 180 ry 0 rz -180 deg; joints [-136.323, -41.96, -99.396, 50.717, 63.15, -28.905]
  MoveL 10989 to (-40.32, 47.93, 153.89) mm, rotated rx 180 ry 0 rz -180 deg; joints [-136.323, -41.96, -99.396, 50.717, 63.15, -28.905]
  Call Extruder(62.24897)
  MoveL 10990 to (-40.27, 47.68, 153.89) mm, rotated rx 180 ry 0 rz 180 deg; joints [-136.358, -41.95, -99.42, 50.678, 63.142, -28.878]
  MoveL 10991 to (-40.27, 47.68, 153.89) mm, rotated rx 180 ry 0 rz 180 deg; joints [-136.358, -41.95, -99.42, 50.678, 63.142, -28.878]
  Call Extruder(62.38656)
  MoveL 10992 to (-40.22, 47.43, 153.89) mm, rotated rx -180 ry 0 rz 180 deg; joints [-136.393, -41.94, -99.444, 50.638, 63.134, -28.851]
  MoveL 10993 to (-40.22, 47.43, 153.89) mm, rotated rx -180 ry 0 rz 180 deg; joints [-136.393, -41.94, -99.444, 50.638, 63.134, -28.851]
  Call Extruder(62.50029)
  MoveL 10994 to (-40.17, 47.23, 153.89) mm, rotated rx 180 ry 0 rz -180 deg; joints [-136.422, -41.932, -99.463, 50.605, 63.127, -28.829]
  MoveL 10995 to (-40.17, 47.23, 153.89) mm, rotated rx 180 ry 0 rz -180 deg; joints [-136.422, -41.932, -99.463, 50.605, 63.127, -28.829]
  Call Extruder(62.61447)
  MoveL 10996 to (-40.13, 47.02, 153.89) mm, rotated rx 180 ry 0 rz 180 deg; joints [-136.452, -41.923, -99.482, 50.572, 63.119, -28.806]
  MoveL 10997 to (-40.13, 47.02, 153.89) mm, rotated rx 180 ry 0 rz 180 deg; joints [-136.452, -41.923, -99.482, 50.572, 63.119, -28.806]
  Call Extruder(62.72910)
  MoveL 10998 to (-40.08, 46.82, 153.89) mm, rotated rx 180 ry 0 rz 180 deg; joints [-136.481, -41.915, -99.5, 50.54, 63.112, -28.784]
  MoveL 10999 to (-40.08, 46.82, 153.89) mm, rotated rx 180 ry 0 rz 180 deg; joints [-136.481, -41.915, -99.5, 50.54, 63.112, -28.784]
  Call Extruder(62.84419)
  MoveL 11000 to (-40.04, 46.61, 153.89) mm, rotated rx 180 ry 0 rz 180 deg; joints [-136.51, -41.907, -99.519, 50.507, 63.105, -28.762]
  MoveL 11001 to (-40.04, 46.61, 153.89) mm, rotated rx 180 ry 0 rz 180 deg; joints [-136.51, -41.907, -99.519, 50.507, 63.105, -28.762]
  Call Extruder(62.96643)
  MoveL 11002 to (-39.98, 46.4, 153.89) mm, rotated rx 180 ry 0 rz -180 deg; joints [-136.542, -41.899, -99.538, 50.471, 63.096, -28.738]
  MoveL 11003 to (-39.98, 46.4, 153.89) mm, rotated rx 180 ry 0 rz -180 deg; joints [-136.542, -41.899, -99.538, 50.471, 63.096, -28.738]
  Call Extruder(63.09609)
  MoveL 11004 to (-39.92, 46.18, 153.89) mm, rotated rx 180 ry 0 rz -180 deg; joints [-136.576, -41.892, -99.556, 50.434, 63.087, -28.714]
  MoveL 11005 to (-39.92, 46.18, 153.89) mm, rotated rx 180 ry 0 rz -180 deg; joints [-136.576, -41.892, -99.556, 50.434, 63.087, -28.714]
  Call Extruder(63.22632)
  MoveL 11006 to (-39.85, 45.95, 153.89) mm, rotated rx 180 ry 0 rz 180 deg; joints [-136.61, -41.884, -99.574, 50.396, 63.077, -28.69]
  MoveL 11007 to (-39.85, 45.95, 153.89) mm, rotated rx 180 ry 0 rz 180 deg; joints [-136.61, -41.884, -99.574, 50.396, 63.077, -28.69]
  Call Extruder(63.35712)
  MoveL 11008 to (-39.78, 45.73, 153.89) mm, rotated rx 180 ry 0 rz -180 deg; joints [-136.644, -41.876, -99.592, 50.358, 63.067, -28.666]
  MoveL 11009 to (-39.78, 45.73, 153.89) mm, rotated rx 180 ry 0 rz -180 deg; joints [-136.644, -41.876, -99.592, 50.358, 63.067, -28.666]
  Call Extruder(63.48848)
  MoveL 11010 to (-39.71, 45.51, 153.89) mm, rotated rx 180 ry 0 rz -180 deg; joints [-136.678, -41.868, -99.61, 50.321, 63.057, -28.642]
  MoveL 11011 to (-39.71, 45.51, 153.89) mm, rotated rx 180 ry 0 rz -180 deg; joints [-136.678, -41.868, -99.61, 50.321, 63.057, -28.642]
  Call Extruder(63.60038)
  MoveL 11012 to (-39.65, 45.32, 153.89) mm, rotated rx 180 ry 0 rz -180 deg; joints [-136.707, -41.862, -99.625, 50.289, 63.049, -28.621]
  MoveL 11013 to (-39.65, 45.32, 153.89) mm, rotated rx 180 ry 0 rz -180 deg; joints [-136.707, -41.862, -99.625, 50.289, 63.049, -28.621]
  Call Extruder(63.71272)
  MoveL 11014 to (-39.59, 45.13, 153.89) mm, rotated rx -180 ry 0 rz 180 deg; joints [-136.737, -41.856, -99.64, 50.256, 63.04, -28.601]
  MoveL 11015 to (-39.59, 45.13, 153.89) mm, rotated rx -180 ry 0 rz 180 deg; joints [-136.737, -41.856, -99.64, 50.256, 63.04, -28.601]
  Call Extruder(63.82551)
  MoveL 11016 to (-39.53, 44.94, 153.89) mm, rotated rx 180 ry 0 rz -180 deg; joints [-136.766, -41.85, -99.654, 50.224, 63.031, -28.581]
  MoveL 11017 to (-39.53, 44.94, 153.89) mm, rotated rx 180 ry 0 rz -180 deg; joints [-136.766, -41.85, -99.654, 50.224, 63.031, -28.581]
  Call Extruder(63.93874)
  MoveL 11018 to (-39.47, 44.75, 153.89) mm, rotated rx 180 ry 0 rz -180 deg; joints [-136.796, -41.843, -99.669, 50.192, 63.023, -28.56]
  MoveL 11019 to (-39.47, 44.75, 153.89) mm, rotated rx 180 ry 0 rz -180 deg; joints [-136.796, -41.843, -99.669, 50.192, 63.023, -28.56]
  Call Extruder(64.05242)
  MoveL 11020 to (-39.41, 44.56, 153.89) mm, rotated rx 180 ry 0 rz 180 deg; joints [-136.825, -41.837, -99.684, 50.16, 63.014, -28.54]
  MoveL 11021 to (-39.41, 44.56, 153.89) mm, rotated rx 180 ry 0 rz 180 deg; joints [-136.825, -41.837, -99.684, 50.16, 63.014, -28.54]
  Call Extruder(64.23439)
  MoveL 11022 to (-39.29, 44.27, 153.89) mm, rotated rx -180 ry 0 rz -180 deg; joints [-136.873, -41.829, -99.703, 50.108, 62.998, -28.509]
  MoveL 11023 to (-39.29, 44.27, 153.89) mm, rotated rx -180 ry 0 rz -180 deg; joints [-136.873, -41.829, -99.703, 50.108, 62.998, -28.509]
  Call Extruder(64.41711)
  MoveL 11024 to (-39.16, 43.98, 153.89) mm, rotated rx 180 ry 0 rz -180 deg; joints [-136.922, -41.821, -99.722, 50.056, 62.982, -28.477]
  MoveL 11025 to (-39.16, 43.98, 153.89) mm, rotated rx 180 ry 0 rz -180 deg; joints [-136.922, -41.821, -99.722, 50.056, 62.982, -28.477]
  Call Extruder(64.58752)
  MoveL 11026 to (-39.05, 43.71, 153.89) mm, rotated rx 180 ry 0 rz 180 deg; joints [-136.967, -41.813, -99.74, 50.007, 62.967, -28.449]
  MoveL 11027 to (-39.05, 43.71, 153.89) mm, rotated rx 180 ry 0 rz 180 deg; joints [-136.967, -41.813, -99.74, 50.007, 62.967, -28.449]
  Call Extruder(64.74550)
  MoveL 11028 to (-38.94, 43.46, 153.89) mm, rotated rx 180 ry 0 rz 180 deg; joints [-137.009, -41.806, -99.756, 49.962, 62.953, -28.422]
  MoveL 11029 to (-38.94, 43.46, 153.89) mm, rotated rx 180 ry 0 rz 180 deg; joints [-137.009, -41.806, -99.756, 49.962, 62.953, -28.422]
  Call Extruder(64.90409)
  MoveL 11030 to (-38.84, 43.21, 153.89) mm, rotated rx 180 ry 0 rz 180 deg; joints [-137.05, -41.799, -99.772, 49.917, 62.939, -28.395]
  MoveL 11031 to (-38.84, 43.21, 153.89) mm, rotated rx 180 ry 0 rz 180 deg; joints [-137.05, -41.799, -99.772, 49.917, 62.939, -28.395]
  Call Extruder(65.11025)
  MoveL 11032 to (-38.66, 42.91, 153.89) mm, rotated rx 180 ry 0 rz -180 deg; joints [-137.107, -41.794, -99.786, 49.859, 62.917, -28.363]
  MoveL 11033 to (-38.66, 42.91, 153.89) mm, rotated rx 180 ry 0 rz -180 deg; joints [-137.107, -41.794, -99.786, 49.859, 62.917, -28.363]
  Call Extruder(65.31720)
  MoveL 11034 to (-38.49, 42.6, 153.89) mm, rotated rx -180 ry 0 rz -180 deg; joints [-137.163, -41.788, -99.799, 49.8, 62.896, -28.331]
  MoveL 11035 to (-38.49, 42.6, 153.89) mm, rotated rx -180 ry 0 rz -180 deg; joints [-137.163, -41.788, -99.799, 49.8, 62.896, -28.331]
  Call Extruder(65.52492)
  MoveL 11036 to (-38.31, 42.3, 153.89) mm, rotated rx 180 ry 0 rz 180 deg; joints [-137.219, -41.782, -99.813, 49.742, 62.874, -28.299]
  MoveL 11037 to (-38.31, 42.3, 153.89) mm, rotated rx 180 ry 0 rz 180 deg; joints [-137.219, -41.782, -99.813, 49.742, 62.874, -28.299]
  Call Extruder(65.73342)
  MoveL 11038 to (-38.13, 41.99, 153.89) mm, rotated rx 180 ry 0 rz 180 deg; joints [-137.275, -41.776, -99.826, 49.683, 62.852, -28.267]
  MoveL 11039 to (-38.13, 41.99, 153.89) mm, rotated rx 180 ry 0 rz 180 deg; joints [-137.275, -41.776, -99.826, 49.683, 62.852, -28.267]
  Call Extruder(65.91297)
  MoveL 11040 to (-37.96, 41.75, 153.89) mm, rotated rx 180 ry 0 rz 180 deg; joints [-137.324, -41.774, -99.832, 49.633, 62.832, -28.242]
  MoveL 11041 to (-37.96, 41.75, 153.89) mm, rotated rx 180 ry 0 rz 180 deg; joints [-137.324, -41.774, -99.832, 49.633, 62.832, -28.242]
  Call Extruder(66.24641)
  MoveL 11042 to (-37.63, 41.3, 153.89) mm, rotated rx 180 ry 0 rz -180 deg; joints [-137.415, -41.769, -99.844, 49.541, 62.793, -28.196]
  MoveL 11043 to (-37.63, 41.3, 153.89) mm, rotated rx 180 ry 0 rz -180 deg; joints [-137.415, -41.769, -99.844, 49.541, 62.793, -28.196]
  Call Extruder(66.58104)
  MoveL 11044 to (-37.3, 40.85, 153.89) mm, rotated rx -180 ry 0 rz 180 deg; joints [-137.506, -41.764, -99.855, 49.448, 62.754, -28.149]
  Call Extruder(67.40900)
  MoveL 11045 to (-36.39, 39.81, 153.89) mm, rotated rx 180 ry 0 rz -180 deg; joints [-137.733, -41.762, -99.859, 49.222, 62.649, -28.043]
  Call Extruder(68.06491)
  MoveL 11046 to (-35.57, 39.08, 153.89) mm, rotated rx 180 ry 0 rz -180 deg; joints [-137.911, -41.771, -99.838, 49.049, 62.557, -27.972]
  Call Extruder(68.40395)
  MoveL 11047 to (-35.13, 38.73, 153.89) mm, rotated rx 180 ry 0 rz 180 deg; joints [-138.003, -41.778, -99.822, 48.962, 62.508, -27.938]
  MoveL 11048 to (-35.13, 38.73, 153.89) mm, rotated rx 180 ry 0 rz 180 deg; joints [-138.003, -41.778, -99.822, 48.962, 62.508, -27.938]
  Call Extruder(68.73731)
  MoveL 11049 to (-34.68, 38.41, 153.89) mm, rotated rx 180 ry 0 rz 180 deg; joints [-138.092, -41.787, -99.801, 48.877, 62.458, -27.907]
  MoveL 11050 to (-34.68, 38.41, 153.89) mm, rotated rx 180 ry 0 rz 180 deg; joints [-138.092, -41.787, -99.801, 48.877, 62.458, -27.907]
  Call Extruder(69.06951)
  MoveL 11051 to (-34.22, 38.08, 153.89) mm, rotated rx 180 ry 0 rz 180 deg; joints [-138.182, -41.796, -99.781, 48.793, 62.409, -27.875]
  MoveL 11052 to (-34.22, 38.08, 153.89) mm, rotated rx 180 ry 0 rz 180 deg; joints [-138.182, -41.796, -99.781, 48.793, 62.409, -27.875]
  Call Extruder(69.24304)
  MoveL 11053 to (-33.97, 37.93, 153.89) mm, rotated rx 180 ry 0 rz -180 deg; joints [-138.227, -41.802, -99.765, 48.751, 62.382, -27.862]
  MoveL 11054 to (-33.97, 37.93, 153.89) mm, rotated rx 180 ry 0 rz -180 deg; joints [-138.227, -41.802, -99.765, 48.751, 62.382, -27.862]
  Call Extruder(69.46654)
  MoveL 11055 to (-33.64, 37.74, 153.89) mm, rotated rx 180 ry 0 rz 180 deg; joints [-138.286, -41.811, -99.745, 48.696, 62.346, -27.845]
  MoveL 11056 to (-33.64, 37.74, 153.89) mm, rotated rx 180 ry 0 rz 180 deg; joints [-138.286, -41.811, -99.745, 48.696, 62.346, -27.845]
  Call Extruder(69.68914)
  MoveL 11057 to (-33.32, 37.55, 153.89) mm, rotated rx 180 ry 0 rz -180 deg; joints [-138.345, -41.82, -99.724, 48.642, 62.311, -27.827]
  MoveL 11058 to (-33.32, 37.55, 153.89) mm, rotated rx 180 ry 0 rz -180 deg; joints [-138.345, -41.82, -99.724, 48.642, 62.311, -27.827]
  Call Extruder(69.91084)
  MoveL 11059 to (-32.99, 37.36, 153.89) mm, rotated rx 180 ry 0 rz 180 deg; joints [-138.404, -41.829, -99.703, 48.588, 62.276, -27.81]
  MoveL 11060 to (-32.99, 37.36, 153.89) mm, rotated rx 180 ry 0 rz 180 deg; joints [-138.404, -41.829, -99.703, 48.588, 62.276, -27.81]
  Call Extruder(70.07784)
  MoveL 11061 to (-32.73, 37.25, 153.89) mm, rotated rx -180 ry 0 rz 180 deg; joints [-138.446, -41.838, -99.682, 48.551, 62.248, -27.801]
  MoveL 11062 to (-32.73, 37.25, 153.89) mm, rotated rx -180 ry 0 rz 180 deg; joints [-138.446, -41.838, -99.682, 48.551, 62.248, -27.801]
  Call Extruder(70.24417)
  MoveL 11063 to (-32.46, 37.14, 153.89) mm, rotated rx 180 ry 0 rz 180 deg; joints [-138.488, -41.847, -99.661, 48.513, 62.22, -27.791]
  MoveL 11064 to (-32.46, 37.14, 153.89) mm, rotated rx 180 ry 0 rz 180 deg; joints [-138.488, -41.847, -99.661, 48.513, 62.22, -27.791]
  Call Extruder(70.41418)
  MoveL 11065 to (-32.19, 37.02, 153.89) mm, rotated rx 180 ry 0 rz -180 deg; joints [-138.532, -41.856, -99.639, 48.475, 62.192, -27.782]
  MoveL 11066 to (-32.19, 37.02, 153.89) mm, rotated rx 180 ry 0 rz -180 deg; joints [-138.532, -41.856, -99.639, 48.475, 62.192, -27.782]
  Call Extruder(70.58788)
  MoveL 11067 to (-31.91, 36.91, 153.89) mm, rotated rx 180 ry 0 rz 180 deg; joints [-138.576, -41.866, -99.616, 48.436, 62.162, -27.772]
  MoveL 11068 to (-31.91, 36.91, 153.89) mm, rotated rx 180 ry 0 rz 180 deg; joints [-138.576, -41.866, -99.616, 48.436, 62.162, -27.772]
  Call Extruder(70.76089)
  MoveL 11069 to (-31.64, 36.79, 153.89) mm, rotated rx 180 ry 0 rz -180 deg; joints [-138.62, -41.876, -99.593, 48.397, 62.133, -27.763]
  MoveL 11070 to (-31.64, 36.79, 153.89) mm, rotated rx 180 ry 0 rz -180 deg; joints [-138.62, -41.876, -99.593, 48.397, 62.133, -27.763]
  Call Extruder(70.87435)
  MoveL 11071 to (-31.45, 36.73, 153.89) mm, rotated rx 180 ry 0 rz -180 deg; joints [-138.648, -41.883, -99.576, 48.373, 62.113, -27.758]
  MoveL 11072 to (-31.45, 36.73, 153.89) mm, rotated rx 180 ry 0 rz -180 deg; joints [-138.648, -41.883, -99.576, 48.373, 62.113, -27.758]
  Call Extruder(70.98736)
  MoveL 11073 to (-31.26, 36.67, 153.89) mm, rotated rx 180 ry 0 rz 180 deg; joints [-138.676, -41.891, -99.558, 48.349, 62.094, -27.754]
  MoveL 11074 to (-31.26, 36.67, 153.89) mm, rotated rx 180 ry 0 rz 180 deg; joints [-138.676, -41.891, -99.558, 48.349, 62.094, -27.754]
  Call Extruder(71.09993)
  MoveL 11075 to (-31.07, 36.61, 153.89) mm, rotated rx -180 ry 0 rz 180 deg; joints [-138.704, -41.898, -99.54, 48.325, 62.074, -27.749]
  MoveL 11076 to (-31.07, 36.61, 153.89) mm, rotated rx -180 ry 0 rz 180 deg; joints [-138.704, -41.898, -99.54, 48.325, 62.074, -27.749]
  Call Extruder(71.21206)
  MoveL 11077 to (-30.88, 36.55, 153.89) mm, rotated rx 180 ry 0 rz -180 deg; joints [-138.732, -41.906, -99.523, 48.301, 62.054, -27.744]
  MoveL 11078 to (-30.88, 36.55, 153.89) mm, rotated rx 180 ry 0 rz -180 deg; joints [-138.732, -41.906, -99.523, 48.301, 62.054, -27.744]
  Call Extruder(71.32374)
  MoveL 11079 to (-30.69, 36.49, 153.89) mm, rotated rx 180 ry 0 rz -180 deg; joints [-138.759, -41.913, -99.505, 48.277, 62.035, -27.74]
  MoveL 11080 to (-30.69, 36.49, 153.89) mm, rotated rx 180 ry 0 rz -180 deg; joints [-138.759, -41.913, -99.505, 48.277, 62.035, -27.74]
  Call Extruder(71.45479)
  MoveL 11081 to (-30.47, 36.42, 153.89) mm, rotated rx 180 ry 0 rz 180 deg; joints [-138.792, -41.923, -99.484, 48.25, 62.012, -27.735]
  MoveL 11082 to (-30.47, 36.42, 153.89) mm, rotated rx 180 ry 0 rz 180 deg; joints [-138.792, -41.923, -99.484, 48.25, 62.012, -27.735]
  Call Extruder(71.58528)
  MoveL 11083 to (-30.25, 36.35, 153.89) mm, rotated rx 180 ry 0 rz 180 deg; joints [-138.824, -41.932, -99.462, 48.222, 61.988, -27.73]
  MoveL 11084 to (-30.25, 36.35, 153.89) mm, rotated rx 180 ry 0 rz 180 deg; joints [-138.824, -41.932, -99.462, 48.222, 61.988, -27.73]
  Call Extruder(71.71521)
  MoveL 11085 to (-30.02, 36.28, 153.89) mm, rotated rx -180 ry 0 rz 180 deg; joints [-138.856, -41.941, -99.441, 48.195, 61.965, -27.726]
  MoveL 11086 to (-30.02, 36.28, 153.89) mm, rotated rx -180 ry 0 rz 180 deg; joints [-138.856, -41.941, -99.441, 48.195, 61.965, -27.726]
  Call Extruder(71.84457)
  MoveL 11087 to (-29.8, 36.22, 153.89) mm, rotated rx 180 ry 0 rz -180 deg; joints [-138.889, -41.95, -99.419, 48.167, 61.942, -27.721]
  MoveL 11088 to (-29.8, 36.22, 153.89) mm, rotated rx 180 ry 0 rz -180 deg; joints [-138.889, -41.95, -99.419, 48.167, 61.942, -27.721]
  Call Extruder(71.96654)
  MoveL 11089 to (-29.59, 36.16, 153.89) mm, rotated rx 180 ry 0 rz 180 deg; joints [-138.919, -41.959, -99.397, 48.142, 61.92, -27.717]
  MoveL 11090 to (-29.59, 36.16, 153.89) mm, rotated rx 180 ry 0 rz 180 deg; joints [-138.919, -41.959, -99.397, 48.142, 61.92, -27.717]
  Call Extruder(72.08140)
  MoveL 11091 to (-29.38, 36.12, 153.89) mm, rotated rx -180 ry 0 rz 180 deg; joints [-138.946, -41.969, -99.376, 48.12, 61.899, -27.715]
  MoveL 11092 to (-29.38, 36.12, 153.89) mm, rotated rx -180 ry 0 rz 180 deg; joints [-138.946, -41.969, -99.376, 48.12, 61.899, -27.715]
  Call Extruder(72.19582)
  MoveL 11093 to (-29.18, 36.07, 153.89) mm, rotated rx -180 ry 0 rz 180 deg; joints [-138.973, -41.978, -99.354, 48.097, 61.878, -27.712]
  MoveL 11094 to (-29.18, 36.07, 153.89) mm, rotated rx -180 ry 0 rz 180 deg; joints [-138.973, -41.978, -99.354, 48.097, 61.878, -27.712]
  Call Extruder(72.30978)
  MoveL 11095 to (-28.97, 36.03, 153.89) mm, rotated rx 180 ry 0 rz -180 deg; joints [-139, -41.987, -99.332, 48.075, 61.857, -27.71]
  MoveL 11096 to (-28.97, 36.03, 153.89) mm, rotated rx 180 ry 0 rz -180 deg; joints [-139, -41.987, -99.332, 48.075, 61.857, -27.71]
  Call Extruder(72.42328)
  MoveL 11097 to (-28.77, 35.98, 153.89) mm, rotated rx 180 ry 0 rz -180 deg; joints [-139.028, -41.997, -99.31, 48.052, 61.836, -27.707]
  MoveL 11098 to (-28.77, 35.98, 153.89) mm, rotated rx 180 ry 0 rz -180 deg; joints [-139.028, -41.997, -99.31, 48.052, 61.836, -27.707]
  Call Extruder(72.56057)
  MoveL 11099 to (-28.52, 35.93, 153.89) mm, rotated rx 180 ry 0 rz -180 deg; joints [-139.06, -42.008, -99.283, 48.026, 61.81, -27.705]
  MoveL 11100 to (-28.52, 35.93, 153.89) mm, rotated rx 180 ry 0 rz -180 deg; joints [-139.06, -42.008, -99.283, 48.026, 61.81, -27.705]
  Call Extruder(72.69724)
  MoveL 11101 to (-28.27, 35.88, 153.89) mm, rotated rx 180 ry 0 rz 180 deg; joints [-139.093, -42.02, -99.256, 47.999, 61.785, -27.703]
  MoveL 11102 to (-28.27, 35.88, 153.89) mm, rotated rx 180 ry 0 rz 180 deg; joints [-139.093, -42.02, -99.256, 47.999, 61.785, -27.703]
  Call Extruder(72.83330)
  MoveL 11103 to (-28.02, 35.83, 153.89) mm, rotated rx 180 ry 0 rz -180 deg; joints [-139.126, -42.032, -99.229, 47.973, 61.759, -27.7]
  MoveL 11104 to (-28.02, 35.83, 153.89) mm, rotated rx 180 ry 0 rz -180 deg; joints [-139.126, -42.032, -99.229, 47.973, 61.759, -27.7]
  Call Extruder(72.96875)
  MoveL 11105 to (-27.77, 35.78, 153.89) mm, rotated rx -180 ry 0 rz 180 deg; joints [-139.158, -42.043, -99.202, 47.946, 61.734, -27.698]
  MoveL 11106 to (-27.77, 35.78, 153.89) mm, rotated rx -180 ry 0 rz 180 deg; joints [-139.158, -42.043, -99.202, 47.946, 61.734, -27.698]
  Call Extruder(73.10359)
  MoveL 11107 to (-27.52, 35.73, 153.89) mm, rotated rx 180 ry 0 rz 180 deg; joints [-139.191, -42.055, -99.175, 47.92, 61.708, -27.695]
  MoveL 11108 to (-27.52, 35.73, 153.89) mm, rotated rx 180 ry 0 rz 180 deg; joints [-139.191, -42.055, -99.175, 47.92, 61.708, -27.695]
  Call Extruder(73.23783)
  MoveL 11109 to (-27.27, 35.68, 153.89) mm, rotated rx -180 ry 0 rz -180 deg; joints [-139.223, -42.066, -99.148, 47.893, 61.682, -27.693]
  MoveL 11110 to (-27.27, 35.68, 153.89) mm, rotated rx -180 ry 0 rz -180 deg; joints [-139.223, -42.066, -99.148, 47.893, 61.682, -27.693]
  Call Extruder(73.37145)
  MoveL 11111 to (-27.02, 35.64, 153.89) mm, rotated rx 180 ry 0 rz -180 deg; joints [-139.256, -42.078, -99.12, 47.867, 61.657, -27.691]
  MoveL 11112 to (-27.02, 35.64, 153.89) mm, rotated rx 180 ry 0 rz -180 deg; joints [-139.256, -42.078, -99.12, 47.867, 61.657, -27.691]
  Call Extruder(73.53354)
  MoveL 11113 to (-26.72, 35.59, 153.89) mm, rotated rx -180 ry 0 rz 180 deg; joints [-139.294, -42.093, -99.085, 47.836, 61.626, -27.689]
  MoveL 11114 to (-26.72, 35.59, 153.89) mm, rotated rx -180 ry 0 rz 180 deg; joints [-139.294, -42.093, -99.085, 47.836, 61.626, -27.689]
  Call Extruder(73.69491)
  MoveL 11115 to (-26.41, 35.54, 153.89) mm, rotated rx 180 ry 0 rz 180 deg; joints [-139.332, -42.108, -99.05, 47.806, 61.595, -27.688]
  MoveL 11116 to (-26.41, 35.54, 153.89) mm, rotated rx 180 ry 0 rz 180 deg; joints [-139.332, -42.108, -99.05, 47.806, 61.595, -27.688]
  Call Extruder(73.85555)
  MoveL 11117 to (-26.11, 35.49, 153.89) mm, rotated rx 180 ry 0 rz -180 deg; joints [-139.371, -42.123, -99.015, 47.775, 61.563, -27.686]
  MoveL 11118 to (-26.11, 35.49, 153.89) mm, rotated rx 180 ry 0 rz -180 deg; joints [-139.371, -42.123, -99.015, 47.775, 61.563, -27.686]
  Call Extruder(74.01546)
  MoveL 11119 to (-25.8, 35.44, 153.89) mm, rotated rx 180 ry 0 rz 180 deg; joints [-139.409, -42.138, -98.981, 47.745, 61.532, -27.685]
  MoveL 11120 to (-25.8, 35.44, 153.89) mm, rotated rx 180 ry 0 rz 180 deg; joints [-139.409, -42.138, -98.981, 47.745, 61.532, -27.685]
  Call Extruder(74.17465)
  MoveL 11121 to (-25.5, 35.39, 153.89) mm, rotated rx -180 ry 0 rz -180 deg; joints [-139.447, -42.153, -98.946, 47.714, 61.501, -27.683]
  MoveL 11122 to (-25.5, 35.39, 153.89) mm, rotated rx -180 ry 0 rz -180 deg; joints [-139.447, -42.153, -98.946, 47.714, 61.501, -27.683]
  Call Extruder(74.33311)
  MoveL 11123 to (-25.19, 35.34, 153.89) mm, rotated rx 180 ry 0 rz -180 deg; joints [-139.485, -42.168, -98.91, 47.684, 61.47, -27.682]
  MoveL 11124 to (-25.19, 35.34, 153.89) mm, rotated rx 180 ry 0 rz -180 deg; joints [-139.485, -42.168, -98.91, 47.684, 61.47, -27.682]
  Call Extruder(74.53198)
  MoveL 11125 to (-24.8, 35.3, 153.89) mm, rotated rx 180 ry 0 rz 180 deg; joints [-139.531, -42.188, -98.864, 47.648, 61.431, -27.681]
  MoveL 11126 to (-24.8, 35.3, 153.89) mm, rotated rx 180 ry 0 rz 180 deg; joints [-139.531, -42.188, -98.864, 47.648, 61.431, -27.681]
  Call Extruder(74.72999)
  MoveL 11127 to (-24.42, 35.25, 153.89) mm, rotated rx 180 ry 0 rz 180 deg; joints [-139.577, -42.208, -98.818, 47.612, 61.391, -27.681]
  MoveL 11128 to (-24.42, 35.25, 153.89) mm, rotated rx 180 ry 0 rz 180 deg; joints [-139.577, -42.208, -98.818, 47.612, 61.391, -27.681]
  Call Extruder(74.92713)
  MoveL 11129 to (-24.03, 35.21, 153.89) mm, rotated rx 180 ry 0 rz 180 deg; joints [-139.624, -42.228, -98.772, 47.576, 61.352, -27.681]
  MoveL 11130 to (-24.03, 35.21, 153.89) mm, rotated rx 180 ry 0 rz 180 deg; joints [-139.624, -42.228, -98.772, 47.576, 61.352, -27.681]
  Call Extruder(75.12340)
  MoveL 11131 to (-23.64, 35.16, 153.89) mm, rotated rx 180 ry 0 rz 180 deg; joints [-139.67, -42.248, -98.725, 47.54, 61.313, -27.681]
  MoveL 11132 to (-23.64, 35.16, 153.89) mm, rotated rx 180 ry 0 rz 180 deg; joints [-139.67, -42.248, -98.725, 47.54, 61.313, -27.681]
  Call Extruder(75.36909)
  MoveL 11133 to (-23.15, 35.11, 153.89) mm, rotated rx 180 ry 0 rz 180 deg; joints [-139.726, -42.274, -98.665, 47.497, 61.264, -27.682]
  MoveL 11134 to (-23.15, 35.11, 153.89) mm, rotated rx 180 ry 0 rz 180 deg; joints [-139.726, -42.274, -98.665, 47.497, 61.264, -27.682]
  Call Extruder(75.66381)
  MoveL 11135 to (-22.56, 35.07, 153.89) mm, rotated rx -180 ry 0 rz -180 deg; joints [-139.793, -42.305, -98.592, 47.446, 61.204, -27.685]
  MoveL 11136 to (-22.56, 35.07, 153.89) mm, rotated rx -180 ry 0 rz -180 deg; joints [-139.793, -42.305, -98.592, 47.446, 61.204, -27.685]
  Call Extruder(75.95720)
  MoveL 11137 to (-21.97, 35.02, 153.89) mm, rotated rx 180 ry 0 rz 180 deg; joints [-139.86, -42.337, -98.518, 47.395, 61.145, -27.688]
  MoveL 11138 to (-21.97, 35.02, 153.89) mm, rotated rx 180 ry 0 rz 180 deg; joints [-139.86, -42.337, -98.518, 47.395, 61.145, -27.688]
  Call Extruder(76.39052)
  MoveL 11139 to (-21.1, 34.98, 153.89) mm, rotated rx 180 ry 0 rz 180 deg; joints [-139.956, -42.385, -98.406, 47.324, 61.057, -27.694]
  MoveL 11140 to (-21.1, 34.98, 153.89) mm, rotated rx 180 ry 0 rz 180 deg; joints [-139.956, -42.385, -98.406, 47.324, 61.057, -27.694]
  Call Extruder(76.96268)
  MoveL 11141 to (-19.94, 34.93, 153.89) mm, rotated rx -180 ry 0 rz 180 deg; joints [-140.081, -42.45, -98.255, 47.232, 60.94, -27.705]
  MoveL 11142 to (-19.94, 34.93, 153.89) mm, rotated rx -180 ry 0 rz 180 deg; joints [-140.081, -42.45, -98.255, 47.232, 60.94, -27.705]
  Call Extruder(77.39112)
  MoveL 11143 to (-19.06, 34.91, 153.89) mm, rotated rx 180 ry 0 rz 180 deg; joints [-140.173, -42.5, -98.139, 47.166, 60.853, -27.715]
  Call Extruder(194.20579)
  MoveL 11144 to (219.06, 34.91, 153.89) mm, rotated rx 180 ry 0 rz 180 deg; joints [-155.896, -62.337, -55.839, 43.457, 36.424, -37.323]
  Call Extruder(194.63413)
  MoveL 11145 to (219.94, 34.93, 153.89) mm, rotated rx 180 ry 0 rz 180 deg; joints [-155.931, -62.44, -55.63, 43.509, 36.326, -37.408]
  MoveL 11146 to (219.94, 34.93, 153.89) mm, rotated rx 180 ry 0 rz 180 deg; joints [-155.931, -62.44, -55.63, 43.509, 36.326, -37.408]
  Call Extruder(195.20742)
  MoveL 11147 to (221.1, 34.98, 153.89) mm, rotated rx 180 ry 0 rz -180 deg; joints [-155.975, -62.579, -55.348, 43.584, 36.196, -37.527]
  MoveL 11148 to (221.1, 34.98, 153.89) mm, rotated rx 180 ry 0 rz -180 deg; joints [-155.975, -62.579, -55.348, 43.584, 36.196, -37.527]
  Call Extruder(195.64158)
  MoveL 11149 to (221.97, 35.02, 153.89) mm, rotated rx 180 ry 0 rz 180 deg; joints [-156.007, -62.685, -55.134, 43.644, 36.098, -37.619]
  MoveL 11150 to (221.97, 35.02, 153.89) mm, rotated rx 180 ry 0 rz 180 deg; joints [-156.007, -62.685, -55.134, 43.644, 36.098, -37.619]
  Call Extruder(195.93548)
  MoveL 11151 to (222.56, 35.07, 153.89) mm, rotated rx 180 ry 0 rz 180 deg; joints [-156.026, -62.757, -54.988, 43.687, 36.033, -37.684]
  MoveL 11152 to (222.56, 35.07, 153.89) mm, rotated rx 180 ry 0 rz 180 deg; joints [-156.026, -62.757, -54.988, 43.687, 36.033, -37.684]
  Call Extruder(196.23072)
  MoveL 11153 to (223.15, 35.12, 153.89) mm, rotated rx -180 ry 0 rz 180 deg; joints [-156.046, -62.829, -54.842, 43.731, 35.967, -37.75]
  MoveL 11154 to (223.15, 35.12, 153.89) mm, rotated rx -180 ry 0 rz 180 deg; joints [-156.046, -62.829, -54.842, 43.731, 35.967, -37.75]
  Call Extruder(196.47684)
  MoveL 11155 to (223.64, 35.16, 153.89) mm, rotated rx 180 ry 0 rz 180 deg; joints [-156.062, -62.889, -54.719, 43.769, 35.912, -37.806]
  MoveL 11156 to (223.64, 35.16, 153.89) mm, rotated rx 180 ry 0 rz 180 deg; joints [-156.062, -62.889, -54.719, 43.769, 35.912, -37.806]
  Call Extruder(196.67350)
  MoveL 11157 to (224.03, 35.21, 153.89) mm, rotated rx 180 ry 0 rz -180 deg; joints [-156.074, -62.938, -54.621, 43.801, 35.869, -37.852]
  MoveL 11158 to (224.03, 35.21, 153.89) mm, rotated rx 180 ry 0 rz -180 deg; joints [-156.074, -62.938, -54.621, 43.801, 35.869, -37.852]
  Call Extruder(196.87102)
  MoveL 11159 to (224.42, 35.25, 153.89) mm, rotated rx 180 ry 0 rz 180 deg; joints [-156.085, -62.987, -54.522, 43.833, 35.826, -37.898]
  MoveL 11160 to (224.42, 35.25, 153.89) mm, rotated rx 180 ry 0 rz 180 deg; joints [-156.085, -62.987, -54.522, 43.833, 35.826, -37.898]
  Call Extruder(197.06941)
  MoveL 11161 to (224.8, 35.3, 153.89) mm, rotated rx 180 ry 0 rz -180 deg; joints [-156.097, -63.035, -54.424, 43.865, 35.783, -37.944]
  MoveL 11162 to (224.8, 35.3, 153.89) mm, rotated rx 180 ry 0 rz -180 deg; joints [-156.097, -63.035, -54.424, 43.865, 35.783, -37.944]
  Call Extruder(197.26866)
  MoveL 11163 to (225.19, 35.35, 153.89) mm, rotated rx 180 ry 0 rz 180 deg; joints [-156.109, -63.084, -54.325, 43.897, 35.74, -37.991]
  MoveL 11164 to (225.19, 35.35, 153.89) mm, rotated rx 180 ry 0 rz 180 deg; joints [-156.109, -63.084, -54.325, 43.897, 35.74, -37.991]
  Call Extruder(197.42740)
  MoveL 11165 to (225.5, 35.39, 153.89) mm, rotated rx 180 ry 0 rz 180 deg; joints [-156.117, -63.123, -54.246, 43.925, 35.706, -38.029]
  MoveL 11166 to (225.5, 35.39, 153.89) mm, rotated rx 180 ry 0 rz 180 deg; joints [-156.117, -63.123, -54.246, 43.925, 35.706, -38.029]
  Call Extruder(197.58687)
  MoveL 11167 to (225.8, 35.44, 153.89) mm, rotated rx 180 ry 0 rz 180 deg; joints [-156.125, -63.163, -54.167, 43.953, 35.673, -38.068]
  MoveL 11168 to (225.8, 35.44, 153.89) mm, rotated rx 180 ry 0 rz 180 deg; joints [-156.125, -63.163, -54.167, 43.953, 35.673, -38.068]
  Call Extruder(197.74706)
  MoveL 11169 to (226.11, 35.49, 153.89) mm, rotated rx 180 ry 0 rz 180 deg; joints [-156.133, -63.202, -54.087, 43.981, 35.639, -38.107]
  MoveL 11170 to (226.11, 35.49, 153.89) mm, rotated rx 180 ry 0 rz 180 deg; joints [-156.133, -63.202, -54.087, 43.981, 35.639, -38.107]
  Call Extruder(197.90798)
  MoveL 11171 to (226.41, 35.54, 153.89) mm, rotated rx 180 ry 0 rz 180 deg; joints [-156.141, -63.241, -54.008, 44.01, 35.605, -38.147]
  MoveL 11172 to (226.41, 35.54, 153.89) mm, rotated rx 180 ry 0 rz 180 deg; joints [-156.141, -63.241, -54.008, 44.01, 35.605, -38.147]
  Call Extruder(198.06962)
  MoveL 11173 to (226.72, 35.59, 153.89) mm, rotated rx -180 ry 0 rz 180 deg; joints [-156.149, -63.28, -53.928, 44.038, 35.571, -38.186]
  MoveL 11174 to (226.72, 35.59, 153.89) mm, rotated rx -180 ry 0 rz 180 deg; joints [-156.149, -63.28, -53.928, 44.038, 35.571, -38.186]
  Call Extruder(198.23200)
  MoveL 11175 to (227.02, 35.64, 153.89) mm, rotated rx 180 ry 0 rz 180 deg; joints [-156.156, -63.32, -53.849, 44.066, 35.537, -38.225]
  MoveL 11176 to (227.02, 35.64, 153.89) mm, rotated rx 180 ry 0 rz 180 deg; joints [-156.156, -63.32, -53.849, 44.066, 35.537, -38.225]
  Call Extruder(198.36589)
  MoveL 11177 to (227.27, 35.69, 153.89) mm, rotated rx -180 ry 0 rz 180 deg; joints [-156.162, -63.352, -53.783, 44.091, 35.51, -38.259]
  MoveL 11178 to (227.27, 35.69, 153.89) mm, rotated rx -180 ry 0 rz 180 deg; joints [-156.162, -63.352, -53.783, 44.091, 35.51, -38.259]
  Call Extruder(198.50039)
  MoveL 11179 to (227.52, 35.74, 153.89) mm, rotated rx -180 ry 0 rz 180 deg; joints [-156.168, -63.385, -53.716, 44.116, 35.482, -38.293]
  MoveL 11180 to (227.52, 35.74, 153.89) mm, rotated rx -180 ry 0 rz 180 deg; joints [-156.168, -63.385, -53.716, 44.116, 35.482, -38.293]
  Call Extruder(198.63550)
  MoveL 11181 to (227.77, 35.79, 153.89) mm, rotated rx 180 ry 0 rz 180 deg; joints [-156.173, -63.418, -53.65, 44.141, 35.455, -38.327]
  MoveL 11182 to (227.77, 35.79, 153.89) mm, rotated rx 180 ry 0 rz 180 deg; joints [-156.173, -63.418, -53.65, 44.141, 35.455, -38.327]
  Call Extruder(198.77122)
  MoveL 11183 to (228.02, 35.84, 153.89) mm, rotated rx -180 ry 0 rz -180 deg; joints [-156.179, -63.451, -53.584, 44.167, 35.427, -38.361]
  MoveL 11184 to (228.02, 35.84, 153.89) mm, rotated rx -180 ry 0 rz -180 deg; joints [-156.179, -63.451, -53.584, 44.167, 35.427, -38.361]
  Call Extruder(198.90755)
  MoveL 11185 to (228.27, 35.88, 153.89) mm, rotated rx 180 ry 0 rz 180 deg; joints [-156.184, -63.484, -53.517, 44.192, 35.4, -38.395]
  MoveL 11186 to (228.27, 35.88, 153.89) mm, rotated rx 180 ry 0 rz 180 deg; joints [-156.184, -63.484, -53.517, 44.192, 35.4, -38.395]
  Call Extruder(199.04449)
  MoveL 11187 to (228.52, 35.93, 153.89) mm, rotated rx -180 ry 0 rz 180 deg; joints [-156.19, -63.516, -53.451, 44.218, 35.372, -38.43]
  MoveL 11188 to (228.52, 35.93, 153.89) mm, rotated rx -180 ry 0 rz 180 deg; joints [-156.19, -63.516, -53.451, 44.218, 35.372, -38.43]
  Call Extruder(199.18204)
  MoveL 11189 to (228.77, 35.98, 153.89) mm, rotated rx -180 ry 0 rz -180 deg; joints [-156.195, -63.549, -53.385, 44.243, 35.345, -38.464]
  MoveL 11190 to (228.77, 35.98, 153.89) mm, rotated rx -180 ry 0 rz -180 deg; joints [-156.195, -63.549, -53.385, 44.243, 35.345, -38.464]
  Call Extruder(199.30492)
  MoveL 11191 to (228.99, 36.03, 153.89) mm, rotated rx -180 ry 0 rz 180 deg; joints [-156.2, -63.579, -53.325, 44.267, 35.321, -38.495]
  MoveL 11192 to (228.99, 36.03, 153.89) mm, rotated rx -180 ry 0 rz 180 deg; joints [-156.2, -63.579, -53.325, 44.267, 35.321, -38.495]
  Call Extruder(199.42833)
  MoveL 11193 to (229.21, 36.08, 153.89) mm, rotated rx 180 ry 0 rz -180 deg; joints [-156.204, -63.608, -53.266, 44.29, 35.296, -38.527]
  MoveL 11194 to (229.21, 36.08, 153.89) mm, rotated rx 180 ry 0 rz -180 deg; joints [-156.204, -63.608, -53.266, 44.29, 35.296, -38.527]
  Call Extruder(199.55228)
  MoveL 11195 to (229.43, 36.13, 153.89) mm, rotated rx -180 ry 0 rz 180 deg; joints [-156.209, -63.638, -53.206, 44.314, 35.272, -38.558]
  MoveL 11196 to (229.43, 36.13, 153.89) mm, rotated rx -180 ry 0 rz 180 deg; joints [-156.209, -63.638, -53.206, 44.314, 35.272, -38.558]
  Call Extruder(199.67675)
  MoveL 11197 to (229.65, 36.18, 153.89) mm, rotated rx -180 ry 0 rz -180 deg; joints [-156.213, -63.667, -53.146, 44.337, 35.248, -38.59]
  MoveL 11198 to (229.65, 36.18, 153.89) mm, rotated rx -180 ry 0 rz -180 deg; joints [-156.213, -63.667, -53.146, 44.337, 35.248, -38.59]
  Call Extruder(199.79915)
  MoveL 11199 to (229.86, 36.23, 153.89) mm, rotated rx -180 ry 0 rz -180 deg; joints [-156.217, -63.696, -53.088, 44.362, 35.224, -38.622]
  MoveL 11200 to (229.86, 36.23, 153.89) mm, rotated rx -180 ry 0 rz -180 deg; joints [-156.217, -63.696, -53.088, 44.362, 35.224, -38.622]
  Call Extruder(199.91963)
  MoveL 11201 to (230.07, 36.3, 153.89) mm, rotated rx -180 ry 0 rz -180 deg; joints [-156.219, -63.725, -53.03, 44.388, 35.202, -38.654]
  MoveL 11202 to (230.07, 36.3, 153.89) mm, rotated rx -180 ry 0 rz -180 deg; joints [-156.219, -63.725, -53.03, 44.388, 35.202, -38.654]
  Call Extruder(200.04059)
  MoveL 11203 to (230.28, 36.36, 153.89) mm, rotated rx -180 ry 0 rz -180 deg; joints [-156.222, -63.754, -52.972, 44.413, 35.179, -38.687]
  MoveL 11204 to (230.28, 36.36, 153.89) mm, rotated rx -180 ry 0 rz -180 deg; joints [-156.222, -63.754, -52.972, 44.413, 35.179, -38.687]
  Call Extruder(200.16205)
  MoveL 11205 to (230.49, 36.42, 153.89) mm, rotated rx 180 ry 0 rz -180 deg; joints [-156.224, -63.783, -52.914, 44.439, 35.157, -38.72]
  MoveL 11206 to (230.49, 36.42, 153.89) mm, rotated rx 180 ry 0 rz -180 deg; joints [-156.224, -63.783, -52.914, 44.439, 35.157, -38.72]
  Call Extruder(200.28400)
  MoveL 11207 to (230.69, 36.49, 153.89) mm, rotated rx 180 ry 0 rz 180 deg; joints [-156.227, -63.811, -52.855, 44.464, 35.134, -38.753]
  MoveL 11208 to (230.69, 36.49, 153.89) mm, rotated rx 180 ry 0 rz 180 deg; joints [-156.227, -63.811, -52.855, 44.464, 35.134, -38.753]
  Call Extruder(200.39590)
  MoveL 11209 to (230.88, 36.55, 153.89) mm, rotated rx 180 ry 0 rz 180 deg; joints [-156.229, -63.838, -52.802, 44.488, 35.114, -38.783]
  MoveL 11210 to (230.88, 36.55, 153.89) mm, rotated rx 180 ry 0 rz 180 deg; joints [-156.229, -63.838, -52.802, 44.488, 35.114, -38.783]
  Call Extruder(200.50825)
  MoveL 11211 to (231.07, 36.61, 153.89) mm, rotated rx -180 ry 0 rz 180 deg; joints [-156.231, -63.864, -52.749, 44.513, 35.093, -38.814]
  MoveL 11212 to (231.07, 36.61, 153.89) mm, rotated rx -180 ry 0 rz 180 deg; joints [-156.231, -63.864, -52.749, 44.513, 35.093, -38.814]
  Call Extruder(200.62104)
  MoveL 11213 to (231.26, 36.67, 153.89) mm, rotated rx 180 ry 0 rz 180 deg; joints [-156.233, -63.891, -52.696, 44.537, 35.073, -38.844]
  MoveL 11214 to (231.26, 36.67, 153.89) mm, rotated rx 180 ry 0 rz 180 deg; joints [-156.233, -63.891, -52.696, 44.537, 35.073, -38.844]
  Call Extruder(200.73427)
  MoveL 11215 to (231.45, 36.73, 153.89) mm, rotated rx -180 ry 0 rz 180 deg; joints [-156.235, -63.917, -52.642, 44.561, 35.052, -38.875]
  MoveL 11216 to (231.45, 36.73, 153.89) mm, rotated rx -180 ry 0 rz 180 deg; joints [-156.235, -63.917, -52.642, 44.561, 35.052, -38.875]
  Call Extruder(200.84795)
  MoveL 11217 to (231.64, 36.79, 153.89) mm, rotated rx -180 ry 0 rz 180 deg; joints [-156.237, -63.944, -52.589, 44.585, 35.032, -38.906]
  MoveL 11218 to (231.64, 36.79, 153.89) mm, rotated rx -180 ry 0 rz 180 deg; joints [-156.237, -63.944, -52.589, 44.585, 35.032, -38.906]
  Call Extruder(201.02990)
  MoveL 11219 to (231.93, 36.91, 153.89) mm, rotated rx 180 ry 0 rz 180 deg; joints [-156.238, -63.986, -52.503, 44.628, 35.001, -38.958]
  MoveL 11220 to (231.93, 36.91, 153.89) mm, rotated rx 180 ry 0 rz 180 deg; joints [-156.238, -63.986, -52.503, 44.628, 35.001, -38.958]
  Call Extruder(201.21262)
  MoveL 11221 to (232.22, 37.03, 153.89) mm, rotated rx 180 ry 0 rz 180 deg; joints [-156.238, -64.029, -52.417, 44.67, 34.97, -39.01]
  MoveL 11222 to (232.22, 37.03, 153.89) mm, rotated rx 180 ry 0 rz 180 deg; joints [-156.238, -64.029, -52.417, 44.67, 34.97, -39.01]
  Call Extruder(201.38304)
  MoveL 11223 to (232.49, 37.15, 153.89) mm, rotated rx 180 ry 0 rz 180 deg; joints [-156.239, -64.068, -52.338, 44.71, 34.941, -39.059]
  MoveL 11224 to (232.49, 37.15, 153.89) mm, rotated rx 180 ry 0 rz 180 deg; joints [-156.239, -64.068, -52.338, 44.71, 34.941, -39.059]
  Call Extruder(201.54104)
  MoveL 11225 to (232.74, 37.26, 153.89) mm, rotated rx -180 ry 0 rz 180 deg; joints [-156.239, -64.105, -52.264, 44.747, 34.914, -39.104]
  MoveL 11226 to (232.74, 37.26, 153.89) mm, rotated rx -180 ry 0 rz 180 deg; joints [-156.239, -64.105, -52.264, 44.747, 34.914, -39.104]
  Call Extruder(201.69964)
  MoveL 11227 to (232.99, 37.36, 153.89) mm, rotated rx 180 ry 0 rz -180 deg; joints [-156.239, -64.141, -52.19, 44.785, 34.887, -39.15]
  MoveL 11228 to (232.99, 37.36, 153.89) mm, rotated rx 180 ry 0 rz -180 deg; joints [-156.239, -64.141, -52.19, 44.785, 34.887, -39.15]
  Call Extruder(201.90581)
  MoveL 11229 to (233.29, 37.54, 153.89) mm, rotated rx 180 ry 0 rz 180 deg; joints [-156.236, -64.189, -52.095, 44.838, 34.856, -39.213]
  MoveL 11230 to (233.29, 37.54, 153.89) mm, rotated rx 180 ry 0 rz 180 deg; joints [-156.236, -64.189, -52.095, 44.838, 34.856, -39.213]
  Call Extruder(202.11275)
  MoveL 11231 to (233.6, 37.71, 153.89) mm, rotated rx -180 ry 0 rz 180 deg; joints [-156.232, -64.236, -51.999, 44.892, 34.824, -39.277]
  MoveL 11232 to (233.6, 37.71, 153.89) mm, rotated rx -180 ry 0 rz 180 deg; joints [-156.232, -64.236, -51.999, 44.892, 34.824, -39.277]
  Call Extruder(202.32048)
  MoveL 11233 to (233.9, 37.89, 153.89) mm, rotated rx 180 ry 0 rz 180 deg; joints [-156.228, -64.283, -51.904, 44.946, 34.792, -39.341]
  MoveL 11234 to (233.9, 37.89, 153.89) mm, rotated rx 180 ry 0 rz 180 deg; joints [-156.228, -64.283, -51.904, 44.946, 34.792, -39.341]
  Call Extruder(202.52898)
  MoveL 11235 to (234.21, 38.06, 153.89) mm, rotated rx 180 ry 0 rz 180 deg; joints [-156.224, -64.331, -51.808, 45, 34.761, -39.405]
  MoveL 11236 to (234.21, 38.06, 153.89) mm, rotated rx 180 ry 0 rz 180 deg; joints [-156.224, -64.331, -51.808, 45, 34.761, -39.405]
  Call Extruder(202.70852)
  MoveL 11237 to (234.45, 38.24, 153.89) mm, rotated rx -180 ry 0 rz 180 deg; joints [-156.218, -64.371, -51.727, 45.05, 34.736, -39.462]
  MoveL 11238 to (234.45, 38.24, 153.89) mm, rotated rx -180 ry 0 rz 180 deg; joints [-156.218, -64.371, -51.727, 45.05, 34.736, -39.462]
  Call Extruder(203.04194)
  MoveL 11239 to (234.9, 38.57, 153.89) mm, rotated rx -180 ry 0 rz 180 deg; joints [-156.206, -64.445, -51.578, 45.143, 34.69, -39.569]
  MoveL 11240 to (234.9, 38.57, 153.89) mm, rotated rx -180 ry 0 rz 180 deg; joints [-156.206, -64.445, -51.578, 45.143, 34.69, -39.569]
  Call Extruder(203.37654)
  MoveL 11241 to (235.35, 38.9, 153.89) mm, rotated rx -180 ry 0 rz 180 deg; joints [-156.195, -64.52, -51.427, 45.236, 34.644, -39.676]
  Call Extruder(204.20449)
  MoveL 11242 to (236.39, 39.81, 153.89) mm, rotated rx -180 ry 0 rz 180 deg; joints [-156.154, -64.7, -51.063, 45.481, 34.542, -39.952]
  Call Extruder(205.03243)
  MoveL 11243 to (237.3, 40.85, 153.89) mm, rotated rx -180 ry 0 rz -180 deg; joints [-156.097, -64.873, -50.715, 45.74, 34.456, -40.236]
  Call Extruder(205.19712)
  MoveL 11244 to (237.46, 41.07, 153.89) mm, rotated rx -180 ry 0 rz 180 deg; joints [-156.083, -64.906, -50.649, 45.793, 34.441, -40.293]
  MoveL 11245 to (237.46, 41.07, 153.89) mm, rotated rx -180 ry 0 rz 180 deg; joints [-156.083, -64.906, -50.649, 45.793, 34.441, -40.293]
  Call Extruder(205.52536)
  MoveL 11246 to (237.79, 41.51, 153.89) mm, rotated rx 180 ry 0 rz 180 deg; joints [-156.056, -64.972, -50.516, 45.9, 34.413, -40.408]
  MoveL 11247 to (237.79, 41.51, 153.89) mm, rotated rx 180 ry 0 rz 180 deg; joints [-156.056, -64.972, -50.516, 45.9, 34.413, -40.408]
  Call Extruder(205.85246)
  MoveL 11248 to (238.11, 41.96, 153.89) mm, rotated rx 180 ry 0 rz 180 deg; joints [-156.029, -65.038, -50.384, 46.006, 34.384, -40.523]
  MoveL 11249 to (238.11, 41.96, 153.89) mm, rotated rx 180 ry 0 rz 180 deg; joints [-156.029, -65.038, -50.384, 46.006, 34.384, -40.523]
  Call Extruder(205.98700)
  MoveL 11250 to (238.22, 42.15, 153.89) mm, rotated rx 180 ry 0 rz 180 deg; joints [-156.016, -65.064, -50.332, 46.051, 34.374, -40.571]
  MoveL 11251 to (238.22, 42.15, 153.89) mm, rotated rx 180 ry 0 rz 180 deg; joints [-156.016, -65.064, -50.332, 46.051, 34.374, -40.571]
  Call Extruder(206.20232)
  MoveL 11252 to (238.41, 42.47, 153.89) mm, rotated rx -180 ry 0 rz -180 deg; joints [-155.995, -65.105, -50.25, 46.123, 34.359, -40.647]
  MoveL 11253 to (238.41, 42.47, 153.89) mm, rotated rx -180 ry 0 rz -180 deg; joints [-155.995, -65.105, -50.25, 46.123, 34.359, -40.647]
  Call Extruder(206.41679)
  MoveL 11254 to (238.59, 42.79, 153.89) mm, rotated rx 180 ry 0 rz 180 deg; joints [-155.974, -65.146, -50.167, 46.195, 34.344, -40.723]
  MoveL 11255 to (238.59, 42.79, 153.89) mm, rotated rx 180 ry 0 rz 180 deg; joints [-155.974, -65.146, -50.167, 46.195, 34.344, -40.723]
  Call Extruder(206.63041)
  MoveL 11256 to (238.77, 43.1, 153.89) mm, rotated rx -180 ry 0 rz 180 deg; joints [-155.953, -65.187, -50.085, 46.267, 34.329, -40.8]
  MoveL 11257 to (238.77, 43.1, 153.89) mm, rotated rx -180 ry 0 rz 180 deg; joints [-155.953, -65.187, -50.085, 46.267, 34.329, -40.8]
  Call Extruder(206.80964)
  MoveL 11258 to (238.91, 43.37, 153.89) mm, rotated rx 180 ry 0 rz 180 deg; joints [-155.934, -65.22, -50.018, 46.328, 34.318, -40.864]
  MoveL 11259 to (238.91, 43.37, 153.89) mm, rotated rx 180 ry 0 rz 180 deg; joints [-155.934, -65.22, -50.018, 46.328, 34.318, -40.864]
  Call Extruder(206.95538)
  MoveL 11260 to (239.01, 43.6, 153.89) mm, rotated rx 180 ry 0 rz 180 deg; joints [-155.917, -65.246, -49.966, 46.378, 34.311, -40.915]
  MoveL 11261 to (239.01, 43.6, 153.89) mm, rotated rx 180 ry 0 rz 180 deg; joints [-155.917, -65.246, -49.966, 46.378, 34.311, -40.915]
  Call Extruder(207.10061)
  MoveL 11262 to (239.11, 43.83, 153.89) mm, rotated rx 180 ry 0 rz -180 deg; joints [-155.901, -65.271, -49.914, 46.428, 34.304, -40.967]
  MoveL 11263 to (239.11, 43.83, 153.89) mm, rotated rx 180 ry 0 rz -180 deg; joints [-155.901, -65.271, -49.914, 46.428, 34.304, -40.967]
  Call Extruder(207.28332)
  MoveL 11264 to (239.23, 44.12, 153.89) mm, rotated rx 180 ry 0 rz 180 deg; joints [-155.879, -65.303, -49.85, 46.491, 34.296, -41.033]
  MoveL 11265 to (239.23, 44.12, 153.89) mm, rotated rx 180 ry 0 rz 180 deg; joints [-155.879, -65.303, -49.85, 46.491, 34.296, -41.033]
  Call Extruder(207.46527)
  MoveL 11266 to (239.35, 44.42, 153.89) mm, rotated rx 180 ry 0 rz -180 deg; joints [-155.858, -65.336, -49.785, 46.554, 34.287, -41.098]
  MoveL 11267 to (239.35, 44.42, 153.89) mm, rotated rx 180 ry 0 rz -180 deg; joints [-155.858, -65.336, -49.785, 46.554, 34.287, -41.098]
  Call Extruder(207.61260)
  MoveL 11268 to (239.44, 44.66, 153.89) mm, rotated rx 180 ry 0 rz -180 deg; joints [-155.84, -65.361, -49.734, 46.605, 34.282, -41.151]
  MoveL 11269 to (239.44, 44.66, 153.89) mm, rotated rx 180 ry 0 rz -180 deg; joints [-155.84, -65.361, -49.734, 46.605, 34.282, -41.151]
  Call Extruder(207.72584)
  MoveL 11270 to (239.5, 44.85, 153.89) mm, rotated rx -180 ry 0 rz 180 deg; joints [-155.826, -65.38, -49.696, 46.644, 34.278, -41.191]
  MoveL 11271 to (239.5, 44.85, 153.89) mm, rotated rx -180 ry 0 rz 180 deg; joints [-155.826, -65.38, -49.696, 46.644, 34.278, -41.191]
  Call Extruder(207.83863)
  MoveL 11272 to (239.56, 45.03, 153.89) mm, rotated rx 180 ry 0 rz 180 deg; joints [-155.811, -65.399, -49.659, 46.684, 34.274, -41.231]
  MoveL 11273 to (239.56, 45.03, 153.89) mm, rotated rx 180 ry 0 rz 180 deg; joints [-155.811, -65.399, -49.659, 46.684, 34.274, -41.231]
  Call Extruder(207.95098)
  MoveL 11274 to (239.62, 45.22, 153.89) mm, rotated rx 180 ry 0 rz -180 deg; joints [-155.797, -65.417, -49.621, 46.723, 34.271, -41.272]
  MoveL 11275 to (239.62, 45.22, 153.89) mm, rotated rx 180 ry 0 rz -180 deg; joints [-155.797, -65.417, -49.621, 46.723, 34.271, -41.272]
  Call Extruder(208.06288)
  MoveL 11276 to (239.68, 45.41, 153.89) mm, rotated rx 180 ry 0 rz 180 deg; joints [-155.783, -65.436, -49.584, 46.762, 34.268, -41.312]
  MoveL 11277 to (239.68, 45.41, 153.89) mm, rotated rx 180 ry 0 rz 180 deg; joints [-155.783, -65.436, -49.584, 46.762, 34.268, -41.312]
  Call Extruder(208.18428)
  MoveL 11278 to (239.75, 45.62, 153.89) mm, rotated rx 180 ry 0 rz 180 deg; joints [-155.767, -65.456, -49.543, 46.805, 34.264, -41.356]
  MoveL 11279 to (239.75, 45.62, 153.89) mm, rotated rx 180 ry 0 rz 180 deg; joints [-155.767, -65.456, -49.543, 46.805, 34.264, -41.356]
  Call Extruder(208.31507)
  MoveL 11280 to (239.81, 45.84, 153.89) mm, rotated rx 180 ry 0 rz 180 deg; joints [-155.75, -65.478, -49.499, 46.852, 34.26, -41.403]
  MoveL 11281 to (239.81, 45.84, 153.89) mm, rotated rx 180 ry 0 rz 180 deg; joints [-155.75, -65.478, -49.499, 46.852, 34.26, -41.403]
  Call Extruder(208.44530)
  MoveL 11282 to (239.88, 46.06, 153.89) mm, rotated rx 180 ry 0 rz 180 deg; joints [-155.733, -65.5, -49.456, 46.898, 34.257, -41.45]
  MoveL 11283 to (239.88, 46.06, 153.89) mm, rotated rx 180 ry 0 rz 180 deg; joints [-155.733, -65.5, -49.456, 46.898, 34.257, -41.45]
  Call Extruder(208.57496)
  MoveL 11284 to (239.95, 46.29, 153.89) mm, rotated rx -180 ry 0 rz 180 deg; joints [-155.715, -65.521, -49.412, 46.944, 34.253, -41.498]
  MoveL 11285 to (239.95, 46.29, 153.89) mm, rotated rx -180 ry 0 rz 180 deg; joints [-155.715, -65.521, -49.412, 46.944, 34.253, -41.498]
  Call Extruder(208.70405)
